KUKA KRL program: nutweldroutines.src, nutweldroutines.dat

--- nutweldroutines.src ---
&ACCESS RVO3
&REL 3482
&PARAM DISKPATH = KRC:\R1\TP\NutWeld
DEF NutWeldRoutines( )
   ;*********************************
   ;* Package:     NutWeldRoutines  *
   ;* Release      V1.0.4           *
   ;* Date:        01.2016          *
   ;* GUI Version: > = V8.3         *
   ;*********************************
   ; Declare in NutWeldData.dat Line 460:
   ;DECL REAL rSetUpperLVDT_CLS_W_NUT[3]
   ;rSetUpperLVDT_CLS_W_NUT[1] = 0.0
   ;rSetUpperLVDT_CLS_W_NUT[2] = 0.0
   ;rSetUpperLVDT_CLS_W_NUT[3] = 0.0
   ;DECL REAL rSetLowerLVDT_CLS_W_NUT[3]
   ;rSetLowerLVDT_CLS_W_NUT[1]  = 0.0
   ;rSetLowerLVDT_CLS_W_NUT[2]  = 0.0
   ;rSetLowerLVDT_CLS_W_NUT[3]  = 0.0
   ;DECL BOOL bSaveCurrentValue1=FALSE
   ;DECL BOOL bSaveCurrentValue2=FALSE
   ;DECL BOOL bSaveCurrentValue3=FALSE
END

GLOBAL DEF NutWeld_Bkg( )
   ;FOLD Details
      ;FOLD Declaration
         DECL REAL rPrimaryValue, rSecondaryValue, rSensorSample
         DECL INT nStepCnt
         DECL BOOL bSensorRetry
      ;ENDFOLD (Declaration)
      ;FOLD Implementation
         dopw1_Hidraulyc_Valve = ($PERI_RDY==TRUE)
         dopw2_Hidraulyc_Valve = (($PERI_RDY==TRUE) AND (nMaxGunNr>=2))
         dopw3_Hidraulyc_Valve = (($PERI_RDY==TRUE) AND (nMaxGunNr>=3))
         IF (($EXT==TRUE) AND (bNutWeld_InhibitWeld==TRUE)) THEN
            bNutWeld_InhibitWeld=FALSE ; Weld Inhibit not allowed in Auto
            nNutWeld_Handle_SPS=Set_Krlmsg (#NOTIFY, NutWeld_Msg[60], NutWeld_MsgPar[], NutWeld_MsgOpt_NoStop)
         ENDIF
         ;FOLD Program Reset/Cancel
            IF ((($PRO_STATE1==#P_FREE) OR ($PRO_STATE1==#P_RESET)) AND (bNutWeldProcessReset==FALSE)) THEN
               bNutWeldProcessReset=TRUE
               NutWeld_ProcessReset( )
            ELSE
               IF (($PRO_STATE1<>#P_FREE) AND ($PRO_STATE1<>#P_RESET)) THEN
                  bNutWeldProcessReset=FALSE
               ENDIF
            ENDIF
         ;ENDFOLD (Program Reset/Cancel)
         ;FOLD Status Key Control
            ;FOLD USKB1 - Process Control
               bNutWeldWOJoining = ((($MODE_OP==#EX) AND (di004UseDryCycle==TRUE)) OR ((($MODE_OP==#T1) OR ($MODE_OP==#T2)) AND (bNutWeldWOJoinSTK==TRUE)))
               IF (($MODE_OP==#T1) OR ($MODE_OP==#T2)) THEN
                  IF ((bNutWeldResetSTK==TRUE) AND ($OUT[Get_FaultResetNr(nNutWeldGunNrSTK)]==FALSE)) THEN
                     bNutWeldResetSTK=FALSE
                     PULSE($OUT[Get_FaultResetNr(nNutWeldGunNrSTK)],TRUE,0.25)
                  ENDIF
               ENDIF
            ;ENDFOLD (USKB1 - Process Control)
            ;FOLD USKB2 - Manual Control
               IF (bNutWeldOpnGunSTK==TRUE) THEN
                  dopw_GunWork(nNutWeldGunNrSTK,FALSE)
                  bNutWeldOpnGunSTK=FALSE
               ENDIF
               IF (bNutWeldClsGunSTK==TRUE) THEN
                  dopw_GunWork(nNutWeldGunNrSTK,TRUE)
                  bNutWeldClsGunSTK=FALSE
               ENDIF
               IF (bNutWeldAdvRetPinSTK==TRUE) THEN
                  dopw_PinAdv(nNutWeldGunNrSTK,dipw_PinReturn(nNutWeldGunNrSTK))
                  bNutWeldAdvRetPinSTK=FALSE
               ENDIF
            ;ENDFOLD (USKB2 - Manual Control)
            ;FOLD USKB3-4 Manual NutWeld
               IF ((bNutWeld_ManWeld_Active==TRUE) AND (bNutWeld_ManWeld_Step[20]==TRUE)) THEN
                  bNutWeld_ManWeld_Active=FALSE
                  bNutWeldManWeldSTK=FALSE
                  dopw_GunWork(nNutWeldGunNrSTK,FALSE)
                  dopw_WeldInit(nNutWeldGunNrSTK,FALSE)
                  dopw_NutIntensify(nNutWeldGunNrSTK,FALSE)
                  dopw_StartFeed(nNutWeldGunNrSTK,FALSE)
                  dopw_SetPrgNr(nNutWeldGunNrSTK, 0 )
                  $TIMER_STOP[nNutWeldManWeldTmr]=TRUE
                  FOR nStepCnt=1 to 20
                     bNutWeld_ManWeld_Step[nStepCnt]=FALSE
                  ENDFOR
               ENDIF
               IF ((bNutWeld_ManWeld_Active==TRUE) AND (bNutWeld_ManWeld_Step[11]==TRUE) AND (bNutWeld_ManWeld_Step[12]==FALSE)) THEN
                  ; Open Gun
                  dopw_GunWork(nNutWeldGunNrSTK,FALSE)
                  bNutWeld_ManWeld_Step[20]=TRUE ; Reset Process
               ENDIF
               IF ((bNutWeld_ManWeld_Active==TRUE) AND (bNutWeld_ManWeld_Step[10]==TRUE) AND (bNutWeld_ManWeld_Step[11]==FALSE)) THEN
                  ; Check for Weld Complete
                  IF ($TIMER_FLAG[nNutWeldManWeldTmr]==TRUE) THEN
                     bNutWeld_ManWeld_Step[20]=TRUE ; Reset Process
                     nNutWeld_Handle_SPS=Set_Krlmsg (#NOTIFY, NutWeld_Msg[19], NutWeld_MsgPar[], NutWeld_MsgOpt_NoStop)
                  ELSE
                     IF (dipw_WeldComplete(nNutWeldGunNrSTK)==TRUE) THEN
                        dopw_WeldInit(nNutWeldGunNrSTK,FALSE)
                        dopw_NutIntensify(nNutWeldGunNrSTK,FALSE)
                        bNutWeld_ManWeld_Step[11]=TRUE
                     ENDIF
                  ENDIF
               ENDIF
               IF ((bNutWeld_ManWeld_Active==TRUE) AND (bNutWeld_ManWeld_Step[9]==TRUE) AND (bNutWeld_ManWeld_Step[10]==FALSE)) THEN
                  ; Weld Initiate
                  dopw_WeldInit(nNutWeldGunNrSTK,TRUE)
                  bNutWeld_ManWeld_Step[10]=TRUE
               ENDIF
               IF ((bNutWeld_ManWeld_Active==TRUE) AND (bNutWeld_ManWeld_Step[8]==TRUE) AND (bNutWeld_ManWeld_Step[9]==FALSE)) THEN
                  ; Intensify Gun
                  dopw_NutIntensify(nNutWeldGunNrSTK,TRUE)
                  ; Check for Gun intensified
                  IF ($TIMER_FLAG[nNutWeldManWeldTmr]==TRUE) THEN
                     bNutWeld_ManWeld_Step[20]=TRUE ; Reset Process
                     nNutWeld_Handle_SPS=Set_Krlmsg (#NOTIFY, NutWeld_Msg[18], NutWeld_MsgPar[], NutWeld_MsgOpt_NoStop)
                  ELSE
                     IF (dipw_IntensfPresOk(nNutWeldGunNrSTK)==TRUE) THEN
                        bNutWeld_ManWeld_Step[9]=TRUE
                     ENDIF
                  ENDIF
               ENDIF
               IF ((bNutWeld_ManWeld_Active==TRUE) AND (bNutWeld_ManWeld_Step[7]==TRUE) AND (bNutWeld_ManWeld_Step[8]==FALSE)) THEN
                  ; Check for Nut Present
                  bSensorRetry=FALSE
                  IF (bByPassSmartelec==TRUE) THEN
                     bNutWeld_ManWeld_Step[8]=TRUE
                  ELSE
                     IF ($TIMER_FLAG[nNutWeldManWeldTmr]==TRUE) THEN
                        bNutWeld_ManWeld_Step[20]=TRUE ; Reset Process
                        nNutWeld_Handle_SPS=Set_Krlmsg (#NOTIFY, NutWeld_Msg[nManWeldFault], NutWeld_MsgPar[], NutWeld_MsgOpt_NoStop)
                     ELSE
                        rPrimaryValue = ABS(aiNutSensor(nNutWeldGunNrSTK));
                        WAIT SEC rSensorSettleTime;
                        rSecondaryValue = ABS(aiNutSensor(nNutWeldGunNrSTK));
                        IF (ABS(rPrimaryValue - rSecondaryValue) <= 2) THEN
                           rSensorSample=ABS(aiNutSensor(nNutWeldGunNrSTK))
                           IF ((rSensorSample <= (rNutInvertedValueInUse + rNutSensorTolInUse)) AND (rSensorSample >= (rNutInvertedValueInUse - rNutSensorTolInUse))) THEN
                              nManWeldFault=55
                              bSensorRetry=TRUE
                           ENDIF
                           IF ((rSensorSample <= (rNoNutValueInUse + rNutSensorTolInUse)) AND (rSensorSample >= (rNoNutValueInUse - rNutSensorTolInUse)) AND (bSensorRetry == FALSE)) THEN
                              nManWeldFault=54
                              bSensorRetry=TRUE
                           ENDIF
                           IF ((rSensorSample <= (rNutPresentValueInUse - rNutSensorTol2InUse)) AND (bSensorRetry == FALSE)) THEN
                              nManWeldFault=56
                              bSensorRetry=TRUE
                           ENDIF
                           IF (bSensorRetry==FALSE) THEN
                              nManWeldFault=0
                              bNutWeld_ManWeld_Step[8]=TRUE
                           ENDIF
                        ENDIF
                     ENDIF
                  ENDIF
               ENDIF
               IF ((bNutWeld_ManWeld_Active==TRUE) AND (bNutWeld_ManWeld_Step[6]==TRUE) AND (bNutWeld_ManWeld_Step[7]==FALSE)) THEN
                  ; Check for Gun Closed
                  IF ($TIMER_FLAG[nNutWeldManWeldTmr]==TRUE) THEN
                     bNutWeld_ManWeld_Step[20]=TRUE ; Reset Process
                     nNutWeld_Handle_SPS=Set_Krlmsg (#NOTIFY, NutWeld_Msg[35], NutWeld_MsgPar[], NutWeld_MsgOpt_NoStop)
                  ELSE
                     IF (bpw_GunAtWork(nNutWeldGunNrSTK)==TRUE) THEN
                        bNutWeld_ManWeld_Step[7]=TRUE
                     ENDIF
                  ENDIF
               ENDIF
               IF ((bNutWeld_ManWeld_Active==TRUE) AND (bNutWeld_ManWeld_Step[5]==TRUE) AND (bNutWeld_ManWeld_Step[6]==FALSE)) THEN
                  ; Check for Nut Fed
                  IF ($TIMER_FLAG[nNutWeldManWeldTmr]==TRUE) THEN
                     bNutWeld_ManWeld_Step[20]=TRUE ; Reset Process
                     nNutWeld_Handle_SPS=Set_Krlmsg (#NOTIFY, NutWeld_Msg[49], NutWeld_MsgPar[], NutWeld_MsgOpt_NoStop)
                     dopw_StartFeed(nNutWeldGunNrSTK,FALSE)
                  ELSE
                     IF (dipw_FeedComplt(nNutWeldGunNrSTK)==TRUE) THEN
                        bNutWeld_ManWeld_Step[6]=TRUE
                        ; Close the gun
                        dopw_StartFeed(nNutWeldGunNrSTK,FALSE)
                        dopw_NutIntensify(nNutWeldGunNrSTK,FALSE)
                        dopw_GunWork(nNutWeldGunNrSTK,TRUE)
                     ENDIF
                  ENDIF
               ENDIF
               IF ((bNutWeld_ManWeld_Active==TRUE) AND (bNutWeld_ManWeld_Step[4]==TRUE) AND (bNutWeld_ManWeld_Step[5]==FALSE)) THEN
                  ; Feed a Nut
                  dopw_StartFeed(nNutWeldGunNrSTK,TRUE)
                  bNutWeld_ManWeld_Step[5]=TRUE
               ENDIF
               IF ((bNutWeld_ManWeld_Active==TRUE) AND (bNutWeld_ManWeld_Step[3]==TRUE) AND (bNutWeld_ManWeld_Step[4]==FALSE)) THEN
                  ; Check for start conditions
                  IF (dipw_XtfmrTempOk(nNutWeldGunNrSTK)==FALSE) THEN
                     bNutWeld_ManWeld_Step[20]=TRUE ; Reset Process
                     nNutWeld_Handle_SPS=Set_Krlmsg (#NOTIFY, NutWeld_Msg[50], NutWeld_MsgPar[], NutWeld_MsgOpt_NoStop)
                  ENDIF
                  IF (dipw_WaterOk(nNutWeldGunNrSTK)==FALSE) THEN
                     bNutWeld_ManWeld_Step[20]=TRUE ; Reset Process
                     nNutWeld_Handle_SPS=Set_Krlmsg (#NOTIFY, NutWeld_Msg[5], NutWeld_MsgPar[], NutWeld_MsgOpt_NoStop)
                  ENDIF
                  IF (dipw_IntensfPresOk(nNutWeldGunNrSTK)==TRUE) THEN
                     bNutWeld_ManWeld_Step[20]=TRUE ; Reset Process
                     nNutWeld_Handle_SPS=Set_Krlmsg (#NOTIFY, NutWeld_Msg[7], NutWeld_MsgPar[], NutWeld_MsgOpt_NoStop)
                  ENDIF
                  IF (dipw_Ready(nNutWeldGunNrSTK)==FALSE) THEN
                     bNutWeld_ManWeld_Step[20]=TRUE ; Reset Process
                     nNutWeld_Handle_SPS=Set_Krlmsg (#NOTIFY, NutWeld_Msg[8], NutWeld_MsgPar[], NutWeld_MsgOpt_NoStop)
                  ENDIF
                  IF (dipw_Fault(nNutWeldGunNrSTK)==TRUE) THEN
                     bNutWeld_ManWeld_Step[20]=TRUE ; Reset Process
                     nNutWeld_Handle_SPS=Set_Krlmsg (#NOTIFY, NutWeld_Msg[9], NutWeld_MsgPar[], NutWeld_MsgOpt_NoStop)
                  ENDIF
                  IF (dipw_SpearHome(nNutWeldGunNrSTK)==FALSE) THEN
                     bNutWeld_ManWeld_Step[20]=TRUE ; Reset Process
                     nNutWeld_Handle_SPS=Set_Krlmsg (#NOTIFY, NutWeld_Msg[47], NutWeld_MsgPar[], NutWeld_MsgOpt_NoStop)
                  ENDIF
                  IF (dipw_PinReturn(nNutWeldGunNrSTK)==FALSE) THEN
                     bNutWeld_ManWeld_Step[20]=TRUE ; Reset Process
                     nNutWeld_Handle_SPS=Set_Krlmsg (#NOTIFY, NutWeld_Msg[15], NutWeld_MsgPar[], NutWeld_MsgOpt_NoStop)
                  ENDIF
                  IF (bpw_GunAtHome(nNutWeldGunNrSTK)==FALSE) THEN
                     bNutWeld_ManWeld_Step[20]=TRUE ; Reset Process
                     nNutWeld_Handle_SPS=Set_Krlmsg (#NOTIFY, NutWeld_Msg[51], NutWeld_MsgPar[], NutWeld_MsgOpt_NoStop)
                  ENDIF
                  bNutWeld_ManWeld_Step[4]=TRUE
               ENDIF
               IF ((bNutWeld_ManWeld_Active==TRUE) AND (bNutWeld_ManWeld_Step[2]==TRUE) AND (bNutWeld_ManWeld_Step[3]==FALSE)) THEN
                  IF (Exists_KrlDlg(nNutWeld_MWHandle, nNutWeld_MWKey)==FALSE) THEN
                     IF (nNutWeld_MWKey==1) THEN
                        bNutWeld_ManWeld_Step[3]=TRUE
                        dopw_SetPrgNr(nNutWeldGunNrSTK, nNutWeldSpotNrSTK )
                     ELSE
                        bNutWeld_ManWeld_Step[20]=TRUE ; Reset Process
                     ENDIF
                  ENDIF
                  nNutWeld_MWKey=0
               ENDIF
               IF ((bNutWeld_ManWeld_Active==TRUE) AND (bNutWeld_ManWeld_Step[1]==TRUE) AND (bNutWeld_ManWeld_Step[2]==FALSE)) THEN
                  bNutWeld_ManWeld_Step[2]=TRUE
                  NutWeld_MsgPar[1]={par_type #value, par_int 0}
                  NutWeld_MsgPar[1].par_int=nNutWeldGunNrSTK
                  NutWeld_MsgPar[2]={par_type #value, par_int 0}
                  NutWeld_MsgPar[2].par_int=nNutWeldSpotNrSTK
                  nNutWeld_MWHandle = Set_KrlDlg (NutWeld_Msg[34], NutWeld_MsgPar[], NutWeld_SK_OKCancel[], NutWeld_MsgOpt_NoStop)
               ENDIF
               IF ((bNutWeldManWeldSTK==TRUE) AND (bNutWeld_ManWeld_Step[1]==FALSE)) THEN
                  IF (bNutWeldWOJoining==FALSE) THEN
                     bNutWeld_ManWeld_Active=TRUE
                     bNutWeld_ManWeld_Step[1]=TRUE
                     dopw_GunWork(nNutWeldGunNrSTK,FALSE)
                     dopw_StartFeed(nNutWeldGunNrSTK,FALSE)
                     dopw_WeldInit(nNutWeldGunNrSTK,FALSE)
                     dopw_NutIntensify(nNutWeldGunNrSTK,FALSE)
                     NutWeldManual.GunNr=nNutWeldGunNrSTK
                     NutWeldManual.SpotNr=nNutWeldSpotNrSTK
                     PWInitUserIO(NutWeldManual)
                     $TIMER_STOP[nNutWeldManWeldTmr]=TRUE
                     $TIMER[nNutWeldManWeldTmr]=(nNutWeld_ManWeld_Timeout*(-1000))
                     $TIMER_STOP[nNutWeldManWeldTmr]=FALSE
                  ELSE
                     nNutWeld_Handle_SPS=Set_Krlmsg (#NOTIFY, NutWeld_Msg[33], NutWeld_MsgPar[], NutWeld_MsgOpt_NoStop)
                     bNutWeldManWeldSTK=FALSE
                  ENDIF
               ENDIF
            ;ENDFOLD (USKB3-4 Manual NutWeld)
            ;FOLD USKB4 - Gun Maintenance Actions
               ;FOLD USKB4-2 Test Gun Force
                  IF ((bNutWeld_TstFrce_Active==TRUE) AND (bNutWeld_TstFrce_Step[10]==TRUE)) THEN
                     bNutWeld_TstFrce_Active=FALSE
                     bNutWeldTstFrceSTK=FALSE
                     dopw_GunWork(nNutWeldGunNrSTK,FALSE)
                     dopw_WeldInit(nNutWeldGunNrSTK,FALSE)
                     dopw_NutIntensify(nNutWeldGunNrSTK,FALSE)
                     dopw_SetPrgNr(nNutWeldGunNrSTK, 0)
                     $TIMER_STOP[nNutWeldManWeldTmr]=TRUE
                     $TIMER_STOP[nNutWeldSignalTmr]=TRUE
                     $TIMER[nNutWeldManWeldTmr]=-1000
                     $TIMER[nNutWeldSignalTmr]=-750
                     FOR nStepCnt=1 to 10
                        bNutWeld_TstFrce_Step[nStepCnt]=FALSE
                     ENDFOR
                  ENDIF
                  IF ((bNutWeld_TstFrce_Active==TRUE) AND (bNutWeld_TstFrce_Step[6]==TRUE) AND (bNutWeld_TstFrce_Step[7]==FALSE)) THEN
                     ; Wait Intensify Time
                     IF ($TIMER_FLAG[nNutWeldSignalTmr]==TRUE) THEN
                        $TIMER_STOP[nNutWeldSignalTmr]=TRUE
                        $TIMER[nNutWeldSignalTmr]=(-2000)
                        dopw_NutIntensify(nNutWeldGunNrSTK,FALSE)
                        dopw_GunWork(nNutWeldGunNrSTK,FALSE)
                        bNutWeld_TstFrce_Step[10]=TRUE
                        NutWeld_MsgPar[1]={par_type #value, par_int 0}
                        NutWeld_MsgPar[1].par_int=nNutWeldGunNrSTK
                        nNutWeld_Handle_SPS=Set_Krlmsg (#NOTIFY, NutWeld_Msg[44], NutWeld_MsgPar[], NutWeld_MsgOpt_NoStop)
                     ENDIF
                  ENDIF
                  IF ((bNutWeld_TstFrce_Active==TRUE) AND (bNutWeld_TstFrce_Step[5]==TRUE) AND (bNutWeld_TstFrce_Step[6]==FALSE)) THEN
                     ; Check for Gun Closed
                     IF (($TIMER_FLAG[nNutWeldManWeldTmr]==TRUE) AND (bpw_GunAtHome(nNutWeldGunNrSTK)==TRUE)) THEN
                        bNutWeld_TstFrce_Step[10]=TRUE ; Reset Process
                        nNutWeld_Handle_SPS=Set_Krlmsg (#NOTIFY, NutWeld_Msg[35], NutWeld_MsgPar[], NutWeld_MsgOpt_NoStop)
                     ELSE
                        IF (($TIMER_FLAG[nNutWeldSignalTmr]==TRUE) AND (bpw_GunAtHome(nNutWeldGunNrSTK)==FALSE)) THEN
                           ; Intensify Gun
                           dopw_NutIntensify(nNutWeldGunNrSTK,TRUE)
                           $TIMER_STOP[nNutWeldSignalTmr]=TRUE
                           $TIMER[nNutWeldSignalTmr]=(-2000)
                           $TIMER_STOP[nNutWeldSignalTmr]=FALSE
                           bNutWeld_TstFrce_Step[6]=TRUE
                        ENDIF
                     ENDIF
                  ENDIF
                  IF ((bNutWeld_TstFrce_Active==TRUE) AND (bNutWeld_TstFrce_Step[4]==TRUE) AND (bNutWeld_TstFrce_Step[5]==FALSE)) THEN
                     IF (Exists_KrlDlg(nNutWeld_TFHandle, nNutWeld_TFKey)==FALSE) THEN
                        IF (nNutWeld_TFKey==1) THEN
                           $TIMER_STOP[nNutWeldManWeldTmr]=FALSE
                           dopw_NutIntensify(nNutWeldGunNrSTK,FALSE)
                           dopw_GunWork(nNutWeldGunNrSTK,TRUE)
                           $TIMER_STOP[nNutWeldSignalTmr]=TRUE
                           $TIMER[nNutWeldSignalTmr]=(-2000)
                           $TIMER_STOP[nNutWeldSignalTmr]=FALSE
                           bNutWeld_TstFrce_Step[5]=TRUE
                        ELSE
                           bNutWeld_TstFrce_Step[10]=TRUE ; Reset Process
                        ENDIF
                     ENDIF
                     nNutWeld_TFKey=0
                  ENDIF
                  IF ((bNutWeldTstFrceSTK==TRUE) AND (bNutWeld_TstFrce_Step[3]==TRUE) AND (bNutWeld_TstFrce_Step[4]==FALSE)) THEN
                     bNutWeld_TstFrce_Active=TRUE
                     bNutWeld_TstFrce_Step[4]=TRUE
                     $TIMER_STOP[nNutWeldManWeldTmr]=TRUE
                     $TIMER[nNutWeldManWeldTmr]=(nNutWeld_ManWeld_Timeout*(-1000))
                     nNutWeld_TFKey=0
                     NutWeld_MsgPar[1]={par_type #value, par_int 0}
                     NutWeld_MsgPar[1].par_int=nNutWeldGunNrSTK
                     nNutWeld_TFHandle = Set_KrlDlg (NutWeld_Msg[38], NutWeld_MsgPar[], NutWeld_SK_TstCncl[], NutWeld_MsgOpt_NoStop)
                  ENDIF
                  IF ((bNutWeld_TstFrce_Active==TRUE) AND (bNutWeld_TstFrce_Step[2]==TRUE) AND (bNutWeld_TstFrce_Step[3]==FALSE)) THEN
                     ; Check for Gun Home
                     IF ($TIMER_FLAG[nNutWeldManWeldTmr]==TRUE) THEN
                        bNutWeld_TstFrce_Step[10]=TRUE ; Reset Process
                        nNutWeld_Handle_SPS=Set_Krlmsg (#NOTIFY, NutWeld_Msg[32], NutWeld_MsgPar[], NutWeld_MsgOpt_NoStop)
                     ELSE
                        IF (($TIMER_FLAG[nNutWeldSignalTmr]==FALSE) AND (bpw_GunAtHome(nNutWeldGunNrSTK)==TRUE)) THEN
                           ; Intensify Gun
                           $TIMER_STOP[nNutWeldSignalTmr]=TRUE
                           $TIMER[nNutWeldSignalTmr]=(-2000)
                           bNutWeld_TstFrce_Step[3]=TRUE
                        ENDIF
                     ENDIF
                  ENDIF
                  IF ((bNutWeld_TstFrce_Active==TRUE) AND (bNutWeld_TstFrce_Step[1]==TRUE) AND (bNutWeld_TstFrce_Step[2]==FALSE)) THEN
                     IF (Exists_KrlDlg(nNutWeld_TFHandle, nNutWeld_TFKey)==FALSE) THEN
                        IF (nNutWeld_TFKey==1) THEN
                           dopw_NutIntensify(nNutWeldGunNrSTK,FALSE)
                           dopw_GunWork(nNutWeldGunNrSTK,FALSE)
                           $TIMER_STOP[nNutWeldSignalTmr]=TRUE
                           $TIMER[nNutWeldSignalTmr]=(-3000)
                           $TIMER_STOP[nNutWeldSignalTmr]=FALSE
                           bNutWeld_TstFrce_Step[2]=TRUE
                        ELSE
                           bNutWeld_TstFrce_Step[10]=TRUE ; Reset Process
                        ENDIF
                     ENDIF
                     nNutWeld_TFKey=0
                  ENDIF
                  IF ((bNutWeldTstFrceSTK==TRUE) AND (bNutWeld_TstFrce_Step[1]==FALSE) AND (bpw_GunAtHome(nNutWeldGunNrSTK )==TRUE)) THEN
                     bNutWeld_TstFrce_Active=TRUE
                     bNutWeld_TstFrce_Step[1]=TRUE
                     bNutWeld_TstFrce_Step[2]=TRUE
                     bNutWeld_TstFrce_Step[3]=TRUE
                     nNutWeld_TFKey=0
                  ELSE
                     IF ((bNutWeldTstFrceSTK==TRUE) AND (bNutWeld_TstFrce_Step[1]==FALSE) AND (bpw_GunAtHome(nNutWeldGunNrSTK )==FALSE)) THEN
                        bNutWeld_TstFrce_Active=TRUE
                        bNutWeld_TstFrce_Step[1]=TRUE
                        nNutWeld_TFKey=0
                        NutWeld_MsgPar[1]={par_type #value, par_int 0}
                        NutWeld_MsgPar[1].par_int=nNutWeldGunNrSTK
                        nNutWeld_TFHandle = Set_KrlDlg (NutWeld_Msg[51], NutWeld_MsgPar[], NutWeld_SK_HomeGun[], NutWeld_MsgOpt_NoStop)
                        $TIMER_STOP[nNutWeldManWeldTmr]=TRUE
                        $TIMER[nNutWeldManWeldTmr]=(nNutWeld_ManWeld_Timeout*(-1000))
                     ENDIF
                  ENDIF
               ;ENDFOLD (USKB4-2 Test Gun Force)
               ;FOLD USKB4-3 Teach Analog
                  ;FOLD USKB4-2.4 Check
                     IF ((bNutWeld_AlgCheck_Active==TRUE) AND (bNutWeld_AlgCheck_Step[10]==TRUE)) THEN
                        bNutWeld_AlgCheck_Active=FALSE
                        bNutWeldAlgCheckReq=FALSE
                        FOR nStepCnt=1 to 10
                           bNutWeld_AlgCheck_Step[nStepCnt]=FALSE
                        ENDFOR
                        bNutWeld_TchAnlg_Active=FALSE
                        bNutWeldTchAnlgSTK=TRUE
                        FOR nStepCnt=1 to 10
                           bNutWeld_TchAnlg_Step[nStepCnt]=FALSE
                        ENDFOR
                     ENDIF
                     IF ((bNutWeld_AlgCheck_Active==TRUE) AND (bNutWeld_AlgCheck_Step[8]==TRUE) AND (bNutWeld_AlgCheck_Step[9]==FALSE)) THEN
                        IF (Exists_KrlDlg(nNutWeld_TA4Handle, nNutWeld_TA4Key)==FALSE) THEN
                           IF (nNutWeld_TA4Key==1) THEN
                              nNutWeld_TA4Key=0
                              bNutWeld_AlgCheck_Step[9]=TRUE
                              bNutWeld_AlgCheck_Step[10]=TRUE
                           ELSE
                              bNutWeld_AlgCheck_Step[10]=TRUE ; Reset Process
                           ENDIF
                        ENDIF
                        nNutWeld_TA4Key=0
                     ENDIF
                     IF ((bNutWeld_AlgCheck_Active==TRUE) AND (bNutWeld_AlgCheck_Step[7]==TRUE) AND (bNutWeld_AlgCheck_Step[8]==FALSE)) THEN
                        IF (rNutInvertedValue[nNutWeldGunNrSTK] < (rNutPresentValue[nNutWeldGunNrSTK] + rNutSensorTolerance[nNutWeldGunNrSTK])) THEN
                           nNutWeld_TA4Handle = Set_KrlDlg (NutWeld_Msg[59], NutWeld_MsgPar[], NutWeld_SK_Next[], NutWeld_MsgOpt_NoStop)
                           bNutWeld_AlgCheck_Step[8]=TRUE
                        ELSE
                           bNutWeld_AlgCheck_Step[10]=TRUE
                        ENDIF
                     ENDIF
                     IF ((bNutWeld_AlgCheck_Active==TRUE) AND (bNutWeld_AlgCheck_Step[6]==TRUE) AND (bNutWeld_AlgCheck_Step[7]==FALSE)) THEN
                        IF (Exists_KrlDlg(nNutWeld_TA4Handle, nNutWeld_TA4Key)==FALSE) THEN
                           IF (nNutWeld_TA4Key==1) THEN
                              nNutWeld_TA4Key=0
                              bNutWeld_AlgCheck_Step[7]=TRUE
                           ELSE
                              bNutWeld_AlgCheck_Step[10]=TRUE ; Reset Process
                           ENDIF
                        ENDIF
                        nNutWeld_TA4Key=0
                     ENDIF
                     IF ((bNutWeld_AlgCheck_Active==TRUE) AND (bNutWeld_AlgCheck_Step[5]==TRUE) AND (bNutWeld_AlgCheck_Step[6]==FALSE)) THEN
                        IF (Exists_KrlDlg(nNutWeld_TA4Handle, nNutWeld_TA4Key)==FALSE) THEN
                           IF (nNutWeld_TA4Key==1) THEN
                              nNutWeld_TA4Key=0
                              bNutWeld_AlgCheck_Step[6]=TRUE
                              IF (rNoNutValue[nNutWeldGunNrSTK] > (rNutPresentValue[nNutWeldGunNrSTK] - rNutSensorTolerance[nNutWeldGunNrSTK])) THEN
                                 nNutWeld_TA4Handle = Set_KrlDlg (NutWeld_Msg[58], NutWeld_MsgPar[], NutWeld_SK_Next[], NutWeld_MsgOpt_NoStop)
                              ELSE
                                 bNutWeld_AlgCheck_Step[7]=TRUE
                              ENDIF
                           ELSE
                              bNutWeld_AlgCheck_Step[10]=TRUE ; Reset Process
                           ENDIF
                        ENDIF
                        nNutWeld_TA4Key=0
                     ENDIF
                     IF ((bNutWeld_AlgCheck_Active==TRUE) AND (bNutWeld_AlgCheck_Step[4]==TRUE) AND (bNutWeld_AlgCheck_Step[5]==FALSE)) THEN
                        IF (Exists_KrlDlg(nNutWeld_TA4Handle, nNutWeld_TA4Key)==FALSE) THEN
                           IF (nNutWeld_TA4Key==1) THEN
                              nNutWeld_TA4Key=0
                              NutWeld_MsgPar[1].par_real=rNutInvertedValue[nNutWeldGunNrSTK]
                              nNutWeld_TA4Handle = Set_KrlDlg (NutWeld_Msg[57], NutWeld_MsgPar[], NutWeld_SK_Next[], NutWeld_MsgOpt_NoStop)
                              bNutWeld_AlgCheck_Step[5]=TRUE
                           ELSE
                              bNutWeld_AlgCheck_Step[10]=TRUE ; Reset Process
                           ENDIF
                        ENDIF
                        nNutWeld_TA4Key=0
                     ENDIF
                     IF ((bNutWeld_AlgCheck_Active==TRUE) AND (bNutWeld_AlgCheck_Step[3]==TRUE) AND (bNutWeld_AlgCheck_Step[4]==FALSE)) THEN
                        IF (Exists_KrlDlg(nNutWeld_TA4Handle, nNutWeld_TA4Key)==FALSE) THEN
                           IF (nNutWeld_TA4Key==1) THEN
                              nNutWeld_TA4Key=0
                              NutWeld_MsgPar[1].par_real=rNutPresentValue[nNutWeldGunNrSTK]
                              nNutWeld_TA4Handle = Set_KrlDlg (NutWeld_Msg[31], NutWeld_MsgPar[], NutWeld_SK_Next[], NutWeld_MsgOpt_NoStop)
                              bNutWeld_AlgCheck_Step[4]=TRUE
                           ELSE
                              bNutWeld_AlgCheck_Step[10]=TRUE ; Reset Process
                           ENDIF
                        ENDIF
                        nNutWeld_TA4Key=0
                     ENDIF
                     IF ((bNutWeld_AlgCheck_Active==TRUE) AND (bNutWeld_AlgCheck_Step[2]==TRUE) AND (bNutWeld_AlgCheck_Step[3]==FALSE)) THEN
                        IF (Exists_KrlDlg(nNutWeld_TA4Handle, nNutWeld_TA4Key)==FALSE) THEN
                           IF (nNutWeld_TA4Key==1) THEN
                              nNutWeld_TA4Key=0
                              NutWeld_MsgPar[1].par_real=rNoNutValue[nNutWeldGunNrSTK]
                              nNutWeld_TA4Handle = Set_KrlDlg (NutWeld_Msg[30], NutWeld_MsgPar[], NutWeld_SK_Next[], NutWeld_MsgOpt_NoStop)
                              bNutWeld_AlgCheck_Step[3]=TRUE
                           ELSE
                              bNutWeld_AlgCheck_Step[10]=TRUE ; Reset Process
                           ENDIF
                        ENDIF
                        nNutWeld_TA4Key=0
                     ENDIF
                     IF ((bNutWeld_AlgCheck_Active==TRUE) AND (bNutWeld_AlgCheck_Step[1]==TRUE) AND (bNutWeld_AlgCheck_Step[2]==FALSE)) THEN
                        IF (Exists_KrlDlg(nNutWeld_TA4Handle, nNutWeld_TA4Key)==FALSE) THEN
                           IF (nNutWeld_TA4Key==1) THEN
                              nNutWeld_TA4Key=0
                              NutWeld_MsgPar[1]={par_type #value, par_real 0}
                              NutWeld_MsgPar[1].par_real=rNutSensorTolerance2[nNutWeldGunNrSTK]
                              nNutWeld_TA4Handle = Set_KrlDlg (NutWeld_Msg[29], NutWeld_MsgPar[], NutWeld_SK_Next[], NutWeld_MsgOpt_NoStop)
                              bNutWeld_AlgCheck_Step[2]=TRUE
                           ELSE
                              bNutWeld_AlgCheck_Step[10]=TRUE ; Reset Process
                           ENDIF
                        ENDIF
                        nNutWeld_TA4Key=0
                     ENDIF
                     IF ((bNutWeldAlgCheckReq==TRUE) AND (bNutWeld_AlgCheck_Step[1]==FALSE)) THEN
                        bNutWeld_AlgCheck_Active=TRUE
                        bNutWeld_AlgCheck_Step[1]=TRUE
                        nNutWeld_TA4Key=0
                        NutWeld_MsgPar[1]={par_type #value, par_real 0}
                        NutWeld_MsgPar[1].par_real=rNutSensorTolerance[nNutWeldGunNrSTK]
                        nNutWeld_TA4Handle = Set_KrlDlg (NutWeld_Msg[28], NutWeld_MsgPar[], NutWeld_SK_Next[], NutWeld_MsgOpt_NoStop)
                     ENDIF
                  ;ENDFOLD (USKB4-2.4 Check)
                  ;FOLD USKB4-2.3 Inverted Nut
                     IF ((bNutWeld_AlgInNut_Active==TRUE) AND (bNutWeld_AlgInNut_Step[10]==TRUE)) THEN
                        bNutWeld_AlgInNut_Active=FALSE
                        bNutWeldAlgInNutReq=FALSE
                        dopw_GunWork(nNutWeldGunNrSTK,FALSE)
                        dopw_NutIntensify(nNutWeldGunNrSTK,FALSE)
                        FOR nStepCnt=1 to 10
                           bNutWeld_AlgInNut_Step[nStepCnt]=FALSE
                        ENDFOR
                        bNutWeld_TchAnlg_Active=FALSE
                        bNutWeldTchAnlgSTK=TRUE
                        $TIMER_STOP[nNutWeldManWeldTmr]=TRUE
                        $TIMER_STOP[nNutWeldSignalTmr]=TRUE
                        $TIMER[nNutWeldManWeldTmr]=-1000
                        $TIMER[nNutWeldSignalTmr]=-750
                        FOR nStepCnt=1 to 10
                           bNutWeld_TchAnlg_Step[nStepCnt]=FALSE
                        ENDFOR
                     ENDIF
                     IF ((bNutWeld_AlgInNut_Active==TRUE) AND (bNutWeld_AlgInNut_Step[6]==TRUE) AND (bNutWeld_AlgInNut_Step[7]==FALSE)) THEN
                        bNutWeld_AlgInNut_Active=FALSE
                        bNutWeldAlgInNutReq=TRUE
                        FOR nStepCnt=1 to 10
                           bNutWeld_AlgInNut_Step[nStepCnt]=FALSE
                        ENDFOR
                     ENDIF
                     IF ((bNutWeld_AlgInNut_Active==TRUE) AND (bNutWeld_AlgInNut_Step[5]==TRUE) AND (bNutWeld_AlgInNut_Step[6]==FALSE)) THEN
                        IF (Exists_KrlDlg(nNutWeld_TA3Handle, nNutWeld_TA3Key)==FALSE) THEN
                           SWITCH nNutWeld_TA3Key
                              CASE 1 ; Accept - Store value and exit
                                 rNutInvertedValue[nNutWeldGunNrSTK]=rNutSensorValueTemp
                                 rNutSensorValueTemp=0.0
                                 bNutWeld_AlgInNut_Step[10]=TRUE ; Reset Process
                              CASE 2 ; Rerun - discard value and re-execute
                                 rNutSensorValueTemp=0.0
                                 bNutWeld_AlgInNut_Step[6]=TRUE ; Local Reset Process
                              CASE 3 ; Cancel - discard value and return to main selection
                                 rNutSensorValueTemp=0.0
                                 bNutWeld_AlgInNut_Step[10]=TRUE ; Reset Process
                           ENDSWITCH
                        ENDIF
                        nNutWeld_TA3Key=0
                     ENDIF
                     IF ((bNutWeld_AlgInNut_Active==TRUE) AND (bNutWeld_AlgInNut_Step[4]==TRUE) AND (bNutWeld_AlgInNut_Step[5]==FALSE)) THEN
                        rNutSensorValueTemp=ABS(aiNutSensor(nNutWeldGunNrSTK))
                        dopw_NutIntensify(nNutWeldGunNrSTK,FALSE)
                        dopw_GunWork(nNutWeldGunNrSTK,FALSE)
                        NutWeld_MsgPar[1]={par_type #value, par_real 0}
                        NutWeld_MsgPar[1].par_real=rNutSensorValueTemp
                        nNutWeld_TA3Handle = Set_KrlDlg (NutWeld_Msg[53], NutWeld_MsgPar[], NutWeld_SK_AcptRerun[], NutWeld_MsgOpt_NoStop)
                        bNutWeld_AlgInNut_Step[5]=TRUE
                     ENDIF
                     IF ((bNutWeld_AlgInNut_Active==TRUE) AND (bNutWeld_AlgInNut_Step[3]==TRUE) AND (bNutWeld_AlgInNut_Step[4]==FALSE)) THEN
                        ; Smart Electrode Dwell Time
                        IF ($TIMER_FLAG[nNutWeldManWeldTmr]==TRUE) THEN
                           $TIMER_STOP[nNutWeldSignalTmr]=TRUE
                           $TIMER[nNutWeldSignalTmr]=(-1000)
                           bNutWeld_AlgInNut_Step[4]=TRUE
                        ENDIF
                     ENDIF
                     IF ((bNutWeld_AlgInNut_Active==TRUE) AND (bNutWeld_AlgInNut_Step[2]==TRUE) AND (bNutWeld_AlgInNut_Step[3]==FALSE)) THEN
                        ; Check for Gun Closed
                        IF ($TIMER_FLAG[nNutWeldManWeldTmr]==TRUE) THEN
                           bNutWeld_AlgInNut_Step[10]=TRUE ; Reset Process
                           nNutWeld_Handle_SPS=Set_Krlmsg (#NOTIFY, NutWeld_Msg[35], NutWeld_MsgPar[], NutWeld_MsgOpt_NoStop)
                        ELSE
                           IF (bpw_GunAtHome(nNutWeldGunNrSTK)==FALSE) THEN
                              $TIMER_STOP[nNutWeldSignalTmr]=TRUE
                              $TIMER[nNutWeldSignalTmr]=(-1000)
                              $TIMER_STOP[nNutWeldSignalTmr]=FALSE
                              bNutWeld_AlgInNut_Step[3]=TRUE
                           ENDIF
                        ENDIF
                     ENDIF
                     IF ((bNutWeld_AlgInNut_Active==TRUE) AND (bNutWeld_AlgInNut_Step[1]==TRUE) AND (bNutWeld_AlgInNut_Step[2]==FALSE)) THEN
                        IF (Exists_KrlDlg(nNutWeld_TA3Handle, nNutWeld_TA3Key)==FALSE) THEN
                           IF (nNutWeld_TA3Key==1) THEN
                              $TIMER_STOP[nNutWeldManWeldTmr]=FALSE
                              dopw_NutIntensify(nNutWeldGunNrSTK,FALSE)
                              dopw_GunWork(nNutWeldGunNrSTK,TRUE)
                              $TIMER_STOP[nNutWeldSignalTmr]=TRUE
                              $TIMER[nNutWeldSignalTmr]=(-750)
                              $TIMER_STOP[nNutWeldSignalTmr]=FALSE
                              bNutWeld_AlgInNut_Step[2]=TRUE
                           ELSE
                              bNutWeld_AlgInNut_Step[10]=TRUE ; Reset Process
                           ENDIF
                        ENDIF
                        nNutWeld_TA3Key=0
                     ENDIF
                     IF ((bNutWeldAlgInNutReq==TRUE) AND (bNutWeld_AlgInNut_Step[1]==FALSE)) THEN
                        bNutWeld_AlgInNut_Active=TRUE
                        bNutWeld_AlgInNut_Step[1]=TRUE
                        dopw_NutIntensify(nNutWeldGunNrSTK,FALSE)
                        dopw_GunWork(nNutWeldGunNrSTK,FALSE)
                        $TIMER_STOP[nNutWeldManWeldTmr]=TRUE
                        $TIMER[nNutWeldManWeldTmr]=(nNutWeld_ManWeld_Timeout*(-1000))
                        $TIMER_STOP[nNutWeldManWeldTmr]=FALSE
                        nNutWeld_TA3Key=0
                        nNutWeld_TA3Handle = Set_KrlDlg (NutWeld_Msg[52], NutWeld_MsgPar[], NutWeld_SK_CloseNWGun[], NutWeld_MsgOpt_NoStop)
                     ENDIF
                  ;ENDFOLD (USKB4-2.3 Inverted Nut)
                  ;FOLD USKB4-2.2 With Nut
                     IF ((bNutWeld_AlgWNut_Active==TRUE) AND (bNutWeld_AlgWNut_Step[10]==TRUE)) THEN
                        bNutWeld_AlgWNut_Active=FALSE
                        bNutWeldAlgWNutReq=FALSE
                        dopw_GunWork(nNutWeldGunNrSTK,FALSE)
                        dopw_NutIntensify(nNutWeldGunNrSTK,FALSE)
                        FOR nStepCnt=1 to 10
                           bNutWeld_AlgWNut_Step[nStepCnt]=FALSE
                        ENDFOR
                        bNutWeld_TchAnlg_Active=FALSE
                        bNutWeldTchAnlgSTK=TRUE
                        $TIMER_STOP[nNutWeldManWeldTmr]=TRUE
                        $TIMER_STOP[nNutWeldSignalTmr]=TRUE
                        $TIMER[nNutWeldManWeldTmr]=-1000
                        $TIMER[nNutWeldSignalTmr]=-750
                        FOR nStepCnt=1 to 10
                           bNutWeld_TchAnlg_Step[nStepCnt]=FALSE
                        ENDFOR
                     ENDIF
                     IF ((bNutWeld_AlgWNut_Active==TRUE) AND (bNutWeld_AlgWNut_Step[6]==TRUE) AND (bNutWeld_AlgWNut_Step[7]==FALSE)) THEN
                        bNutWeld_AlgWNut_Active=FALSE
                        bNutWeldAlgWNutReq=TRUE
                        FOR nStepCnt=1 to 10
                           bNutWeld_AlgWNut_Step[nStepCnt]=FALSE
                        ENDFOR
                     ENDIF
                     IF ((bNutWeld_AlgWNut_Active==TRUE) AND (bNutWeld_AlgWNut_Step[5]==TRUE) AND (bNutWeld_AlgWNut_Step[6]==FALSE)) THEN
                        IF (Exists_KrlDlg(nNutWeld_TA2Handle, nNutWeld_TA2Key)==FALSE) THEN
                           SWITCH nNutWeld_TA2Key
                              CASE 1 ; Accept - Store value and exit
                                 rNutPresentValue[nNutWeldGunNrSTK]=rNutSensorValueTemp
                                 rNutSensorValueTemp=0.0
                                 bNutWeld_AlgWNut_Step[10]=TRUE ; Reset Process
                              CASE 2 ; Rerun - discard value and re-execute
                                 rNutSensorValueTemp=0.0
                                 bNutWeld_AlgWNut_Step[6]=TRUE ; Local Reset Process
                              CASE 3 ; Cancel - discard value and return to main selection
                                 rNutSensorValueTemp=0.0
                                 bNutWeld_AlgWNut_Step[10]=TRUE ; Reset Process
                           ENDSWITCH
                        ENDIF
                        nNutWeld_TA2Key=0
                     ENDIF
                     IF ((bNutWeld_AlgWNut_Active==TRUE) AND (bNutWeld_AlgWNut_Step[4]==TRUE) AND (bNutWeld_AlgWNut_Step[5]==FALSE)) THEN
                        rNutSensorValueTemp=ABS(aiNutSensor(nNutWeldGunNrSTK))
                        dopw_NutIntensify(nNutWeldGunNrSTK,FALSE)
                        dopw_GunWork(nNutWeldGunNrSTK,FALSE)
                        NutWeld_MsgPar[1]={par_type #value, par_real 0}
                        NutWeld_MsgPar[1].par_real=rNutSensorValueTemp
                        nNutWeld_TA2Handle = Set_KrlDlg (NutWeld_Msg[43], NutWeld_MsgPar[], NutWeld_SK_AcptRerun[], NutWeld_MsgOpt_NoStop)
                        bNutWeld_AlgWNut_Step[5]=TRUE
                     ENDIF
                     IF ((bNutWeld_AlgWNut_Active==TRUE) AND (bNutWeld_AlgWNut_Step[3]==TRUE) AND (bNutWeld_AlgWNut_Step[4]==FALSE)) THEN
                        ; Smart Electrode Dwell Time
                        IF ($TIMER_FLAG[nNutWeldManWeldTmr]==TRUE) THEN
                           $TIMER_STOP[nNutWeldSignalTmr]=TRUE
                           $TIMER[nNutWeldSignalTmr]=(-1000)
                           bNutWeld_AlgWNut_Step[4]=TRUE
                        ENDIF
                     ENDIF
                     IF ((bNutWeld_AlgWNut_Active==TRUE) AND (bNutWeld_AlgWNut_Step[2]==TRUE) AND (bNutWeld_AlgWNut_Step[3]==FALSE)) THEN
                        ; Check for Gun Closed
                        IF ($TIMER_FLAG[nNutWeldManWeldTmr]==TRUE) THEN
                           bNutWeld_AlgWNut_Step[10]=TRUE ; Reset Process
                           nNutWeld_Handle_SPS=Set_Krlmsg (#NOTIFY, NutWeld_Msg[35], NutWeld_MsgPar[], NutWeld_MsgOpt_NoStop)
                        ELSE
                           IF (bpw_GunAtHome(nNutWeldGunNrSTK)==FALSE) THEN
                              $TIMER_STOP[nNutWeldSignalTmr]=TRUE
                              $TIMER[nNutWeldSignalTmr]=(-1000)
                              $TIMER_STOP[nNutWeldSignalTmr]=FALSE
                              bNutWeld_AlgWNut_Step[3]=TRUE
                           ENDIF
                        ENDIF
                     ENDIF
                     IF ((bNutWeld_AlgWNut_Active==TRUE) AND (bNutWeld_AlgWNut_Step[1]==TRUE) AND (bNutWeld_AlgWNut_Step[2]==FALSE)) THEN
                        IF (Exists_KrlDlg(nNutWeld_TA2Handle, nNutWeld_TA2Key)==FALSE) THEN
                           IF (nNutWeld_TA2Key==1) THEN
                              $TIMER_STOP[nNutWeldManWeldTmr]=FALSE
                              dopw_NutIntensify(nNutWeldGunNrSTK,FALSE)
                              dopw_GunWork(nNutWeldGunNrSTK,TRUE)
                              $TIMER_STOP[nNutWeldSignalTmr]=TRUE
                              $TIMER[nNutWeldSignalTmr]=(-750)
                              $TIMER_STOP[nNutWeldSignalTmr]=FALSE
                              bNutWeld_AlgWNut_Step[2]=TRUE
                           ELSE
                              bNutWeld_AlgWNut_Step[10]=TRUE ; Reset Process
                           ENDIF
                        ENDIF
                        nNutWeld_TA2Key=0
                     ENDIF
                     IF ((bNutWeldAlgWNutReq==TRUE) AND (bNutWeld_AlgWNut_Step[1]==FALSE)) THEN
                        bNutWeld_AlgWNut_Active=TRUE
                        bNutWeld_AlgWNut_Step[1]=TRUE
                        dopw_NutIntensify(nNutWeldGunNrSTK,FALSE)
                        dopw_GunWork(nNutWeldGunNrSTK,FALSE)
                        $TIMER_STOP[nNutWeldManWeldTmr]=TRUE
                        $TIMER[nNutWeldManWeldTmr]=(nNutWeld_ManWeld_Timeout*(-1000))
                        $TIMER_STOP[nNutWeldManWeldTmr]=FALSE
                        nNutWeld_TA2Key=0
                        nNutWeld_TA2Handle = Set_KrlDlg (NutWeld_Msg[41], NutWeld_MsgPar[], NutWeld_SK_CloseNWGun[], NutWeld_MsgOpt_NoStop)
                     ENDIF
                  ;ENDFOLD (USKB4-2.2 With Nut)
                  ;FOLD USKB4-2.1 No Nut
                     IF ((bNutWeld_AlgNoNut_Active==TRUE) AND (bNutWeld_AlgNoNut_Step[10]==TRUE)) THEN
                        bNutWeld_AlgNoNut_Active=FALSE
                        bNutWeldAlgNoNutReq=FALSE
                        dopw_GunWork(nNutWeldGunNrSTK,FALSE)
                        dopw_NutIntensify(nNutWeldGunNrSTK,FALSE)
                        FOR nStepCnt=1 to 10
                           bNutWeld_AlgNoNut_Step[nStepCnt]=FALSE
                        ENDFOR
                        bNutWeld_TchAnlg_Active=FALSE
                        bNutWeldTchAnlgSTK=TRUE
                        $TIMER_STOP[nNutWeldManWeldTmr]=TRUE
                        $TIMER_STOP[nNutWeldSignalTmr]=TRUE
                        $TIMER[nNutWeldManWeldTmr]=-1000
                        $TIMER[nNutWeldSignalTmr]=-750
                        FOR nStepCnt=1 to 10
                           bNutWeld_TchAnlg_Step[nStepCnt]=FALSE
                        ENDFOR
                     ENDIF
                     IF ((bNutWeld_AlgNoNut_Active==TRUE) AND (bNutWeld_AlgNoNut_Step[6]==TRUE) AND (bNutWeld_AlgNoNut_Step[7]==FALSE)) THEN
                        bNutWeld_AlgNoNut_Active=FALSE
                        bNutWeldAlgNoNutReq=TRUE
                        FOR nStepCnt=1 to 10
                           bNutWeld_AlgNoNut_Step[nStepCnt]=FALSE
                        ENDFOR
                     ENDIF
                     IF ((bNutWeld_AlgNoNut_Active==TRUE) AND (bNutWeld_AlgNoNut_Step[5]==TRUE) AND (bNutWeld_AlgNoNut_Step[6]==FALSE)) THEN
                        IF (Exists_KrlDlg(nNutWeld_TA1Handle, nNutWeld_TA1Key)==FALSE) THEN
                           SWITCH nNutWeld_TA1Key
                              CASE 1 ; Accept - Store value and exit
                                 rNoNutValue[nNutWeldGunNrSTK]=rNutSensorValueTemp
                                 rNutSensorValueTemp=0.0
                                 bNutWeld_AlgNoNut_Step[10]=TRUE ; Reset Process
                              CASE 2 ; Rerun - discard value and re-execute
                                 rNutSensorValueTemp=0.0
                                 bNutWeld_AlgNoNut_Step[6]=TRUE ; Local Reset Process
                              CASE 3 ; Cancel - discard value and return to main selection
                                 rNutSensorValueTemp=0.0
                                 bNutWeld_AlgNoNut_Step[10]=TRUE ; Reset Process
                           ENDSWITCH
                        ENDIF
                        nNutWeld_TA1Key=0
                     ENDIF
                     IF ((bNutWeld_AlgNoNut_Active==TRUE) AND (bNutWeld_AlgNoNut_Step[4]==TRUE) AND (bNutWeld_AlgNoNut_Step[5]==FALSE)) THEN
                        rNutSensorValueTemp=ABS(aiNutSensor(nNutWeldGunNrSTK))
                        dopw_NutIntensify(nNutWeldGunNrSTK,FALSE)
                        dopw_GunWork(nNutWeldGunNrSTK,FALSE)
                        NutWeld_MsgPar[1]={par_type #value, par_real 0}
                        NutWeld_MsgPar[1].par_real=rNutSensorValueTemp
                        nNutWeld_TA1Handle = Set_KrlDlg (NutWeld_Msg[42], NutWeld_MsgPar[], NutWeld_SK_AcptRerun[], NutWeld_MsgOpt_NoStop)
                        bNutWeld_AlgNoNut_Step[5]=TRUE
                     ENDIF
                     IF ((bNutWeld_AlgNoNut_Active==TRUE) AND (bNutWeld_AlgNoNut_Step[3]==TRUE) AND (bNutWeld_AlgNoNut_Step[4]==FALSE)) THEN
                        ; Smart Electrode Dwell Time
                        IF ($TIMER_FLAG[nNutWeldManWeldTmr]==TRUE) THEN
                           $TIMER_STOP[nNutWeldSignalTmr]=TRUE
                           $TIMER[nNutWeldSignalTmr]=(-1000)
                           bNutWeld_AlgNoNut_Step[4]=TRUE
                        ENDIF
                     ENDIF
                     IF ((bNutWeld_AlgNoNut_Active==TRUE) AND (bNutWeld_AlgNoNut_Step[2]==TRUE) AND (bNutWeld_AlgNoNut_Step[3]==FALSE)) THEN
                        ; Check for Gun Closed
                        IF ($TIMER_FLAG[nNutWeldManWeldTmr]==TRUE) THEN
                           bNutWeld_AlgNoNut_Step[10]=TRUE ; Reset Process
                           nNutWeld_Handle_SPS=Set_Krlmsg (#NOTIFY, NutWeld_Msg[35], NutWeld_MsgPar[], NutWeld_MsgOpt_NoStop)
                        ELSE
                           IF (bpw_GunAtHome(nNutWeldGunNrSTK)==FALSE) THEN
                              $TIMER_STOP[nNutWeldSignalTmr]=TRUE
                              $TIMER[nNutWeldSignalTmr]=(-1000)
                              $TIMER_STOP[nNutWeldSignalTmr]=FALSE
                              bNutWeld_AlgNoNut_Step[3]=TRUE
                           ENDIF
                        ENDIF
                     ENDIF
                     IF ((bNutWeld_AlgNoNut_Active==TRUE) AND (bNutWeld_AlgNoNut_Step[1]==TRUE) AND (bNutWeld_AlgNoNut_Step[2]==FALSE)) THEN
                        IF (Exists_KrlDlg(nNutWeld_TA1Handle, nNutWeld_TA1Key)==FALSE) THEN
                           IF (nNutWeld_TA1Key==1) THEN
                              $TIMER_STOP[nNutWeldManWeldTmr]=FALSE
                              dopw_NutIntensify(nNutWeldGunNrSTK,FALSE)
                              dopw_GunWork(nNutWeldGunNrSTK,TRUE)
                              $TIMER_STOP[nNutWeldSignalTmr]=TRUE
                              $TIMER[nNutWeldSignalTmr]=(-750)
                              $TIMER_STOP[nNutWeldSignalTmr]=FALSE
                              bNutWeld_AlgNoNut_Step[2]=TRUE
                           ELSE
                              bNutWeld_AlgNoNut_Step[10]=TRUE ; Reset Process
                           ENDIF
                        ENDIF
                        nNutWeld_TA1Key=0
                     ENDIF
                     IF ((bNutWeldAlgNoNutReq==TRUE) AND (bNutWeld_AlgNoNut_Step[1]==FALSE)) THEN
                        bNutWeld_AlgNoNut_Active=TRUE
                        bNutWeld_AlgNoNut_Step[1]=TRUE
                        dopw_NutIntensify(nNutWeldGunNrSTK,FALSE)
                        dopw_GunWork(nNutWeldGunNrSTK,FALSE)
                        $TIMER_STOP[nNutWeldManWeldTmr]=TRUE
                        $TIMER[nNutWeldManWeldTmr]=(nNutWeld_ManWeld_Timeout*(-1000))
                        $TIMER_STOP[nNutWeldManWeldTmr]=FALSE
                        nNutWeld_TA1Key=0
                        nNutWeld_TA1Handle = Set_KrlDlg (NutWeld_Msg[40], NutWeld_MsgPar[], NutWeld_SK_CloseNWGun[], NutWeld_MsgOpt_NoStop)
                     ENDIF
                  ;ENDFOLD (USKB4-2.1 No Nut)
                  ;FOLD USKB4 Teach Selection
                     IF ((bNutWeld_TchAnlg_Active==TRUE) AND (bNutWeld_TchAnlg_Step[10]==TRUE)) THEN
                        bNutWeld_TchAnlg_Active=FALSE
                        bNutWeldTchAnlgSTK=FALSE
                        dopw_GunWork(nNutWeldGunNrSTK,FALSE)
                        dopw_NutIntensify(nNutWeldGunNrSTK,FALSE)
                        $TIMER_STOP[nNutWeldManWeldTmr]=TRUE
                        $TIMER_STOP[nNutWeldSignalTmr]=TRUE
                        $TIMER[nNutWeldManWeldTmr]=-1000
                        $TIMER[nNutWeldSignalTmr]=-750
                        FOR nStepCnt=1 to 10
                           bNutWeld_TchAnlg_Step[nStepCnt]=FALSE
                        ENDFOR
                     ENDIF
                     IF ((bNutWeld_TchAnlg_Active==TRUE) AND (bNutWeld_TchAnlg_Step[2]==TRUE) AND (bNutWeld_TchAnlg_Step[3]==FALSE)) THEN
                        IF (Exists_KrlDlg(nNutWeld_TAHandle, nNutWeld_TAKey)==FALSE) THEN
                           SWITCH nNutWeld_TAKey
                              CASE 1 ; No Nut
                                 bNutWeldAlgNoNutReq=TRUE
                                 bNutWeld_TchAnlg_Step[3]=TRUE
                              CASE 2 ; With Nut
                                 bNutWeldAlgWNutReq=TRUE
                                 bNutWeld_TchAnlg_Step[3]=TRUE
                              CASE 3 ; Invert Nut
                                 bNutWeldAlgInNutReq=TRUE
                                 bNutWeld_TchAnlg_Step[3]=TRUE
                              CASE 4 ; Check
                                 bNutWeldAlgCheckReq=TRUE
                                 bNutWeld_TchAnlg_Step[3]=TRUE
                              DEFAULT
                                 bNutWeld_TchAnlg_Step[3]=TRUE
                                 bNutWeld_TchAnlg_Step[10]=TRUE ; Reset Process
                           ENDSWITCH
                        ENDIF
                        nNutWeld_TAKey=0
                     ENDIF
                     IF ((bNutWeld_TchAnlg_Active==TRUE) AND (bNutWeld_TchAnlg_Step[1]==TRUE) AND (bNutWeld_TchAnlg_Step[2]==FALSE)) THEN
                        bNutWeld_TchAnlg_Step[2]=TRUE
                        nNutWeld_TAKey=0
                        NutWeld_MsgPar[1]={par_type #value, par_int 0}
                        NutWeld_MsgPar[1].par_int=nNutWeldGunNrSTK
                        nNutWeld_TAHandle = Set_KrlDlg (NutWeld_Msg[39], NutWeld_MsgPar[], NutWeld_SK_TchAnalog[], NutWeld_MsgOpt_NoStop)
                     ENDIF
                     IF ((bNutWeldTchAnlgSTK==TRUE) AND (bNutWeld_TchAnlg_Step[1]==FALSE)) THEN
                        bNutWeld_TchAnlg_Active=TRUE
                        bNutWeld_TchAnlg_Step[1]=TRUE
                     ENDIF
                  ;ENDFOLD (USKB4 Teach Selection)
               ;ENDFOLD (USKB4-4 Teach Analog)
               ;FOLD USKB4-4 Test Welding Current S225
                  IF ((bNutWeld_TstCrnt_Active==TRUE) AND (bNutWeld_TstCrnt_Step[10]==TRUE)) THEN
                     bNutWeld_TstCrnt_Active=FALSE
                     bNutWeldTstCrntSTK=FALSE
                     dopw_GunWork(nNutWeldGunNrSTK,FALSE)
                     dopw_WeldInit(nNutWeldGunNrSTK,FALSE)
                     dopw_NutIntensify(nNutWeldGunNrSTK,FALSE)
                     dopw_SetPrgNr(nNutWeldGunNrSTK, 0)
                     $TIMER_STOP[nNutWeldManWeldTmr]=TRUE
                     $TIMER_STOP[nNutWeldSignalTmr]=TRUE
                     $TIMER[nNutWeldManWeldTmr]=-1000
                     $TIMER[nNutWeldSignalTmr]=-750
                     FOR nStepCnt=1 to 10
                        bNutWeld_TstCrnt_Step[nStepCnt]=FALSE
                     ENDFOR
                  ENDIF
                  IF ((bNutWeld_TstCrnt_Active==TRUE) AND (bNutWeld_TstCrnt_Step[4]==TRUE) AND (bNutWeld_TstCrnt_Step[5]==FALSE)) THEN
                     ; Check for Weld Complete
                     IF ($TIMER_FLAG[nNutWeldManWeldTmr]==TRUE) THEN
                        bNutWeld_TstCrnt_Step[10]=TRUE ; Reset Process
                        nNutWeld_Handle_SPS=Set_Krlmsg (#NOTIFY, NutWeld_Msg[19], NutWeld_MsgPar[], NutWeld_MsgOpt_NoStop)
                     ELSE
                        IF (dipw_WeldComplete(nNutWeldGunNrSTK)==TRUE) THEN
                           dopw_WeldInit(nNutWeldGunNrSTK,FALSE)
                           dopw_NutIntensify(nNutWeldGunNrSTK,FALSE)
                           dopw_GunWork(nNutWeldGunNrSTK,FALSE)
                           bNutWeld_TstCrnt_Step[10]=TRUE
                           nNutWeld_Handle_SPS=Set_Krlmsg (#NOTIFY, NutWeld_Msg[45], NutWeld_MsgPar[], NutWeld_MsgOpt_NoStop)
                        ENDIF
                     ENDIF
                  ENDIF
                  IF ((bNutWeld_TstCrnt_Active==TRUE) AND (bNutWeld_TstCrnt_Step[3]==TRUE) AND (bNutWeld_TstCrnt_Step[4]==FALSE)) THEN
                     ; Check for Gun intensified
                     IF ($TIMER_FLAG[nNutWeldManWeldTmr]==TRUE) THEN
                        bNutWeld_TstCrnt_Step[10]=TRUE ; Reset Process
                        nNutWeld_Handle_SPS=Set_Krlmsg (#NOTIFY, NutWeld_Msg[18], NutWeld_MsgPar[], NutWeld_MsgOpt_NoStop)
                     ELSE
                        IF (dipw_IntensfPresOk(nNutWeldGunNrSTK)==TRUE) THEN
                           bNutWeld_TstCrnt_Step[4]=TRUE
                           dopw_SetPrgNr(nNutWeldGunNrSTK, nSpotNrTstCrnt )
                           ; Weld Initiate
                           dopw_WeldInit(nNutWeldGunNrSTK,TRUE)
                        ENDIF
                     ENDIF
                  ENDIF
                  IF ((bNutWeld_TstCrnt_Active==TRUE) AND (bNutWeld_TstCrnt_Step[2]==TRUE) AND (bNutWeld_TstCrnt_Step[3]==FALSE)) THEN
                     ; Check for Gun Closed
                     IF ($TIMER_FLAG[nNutWeldManWeldTmr]==TRUE) THEN
                        bNutWeld_TstCrnt_Step[10]=TRUE ; Reset Process
                        nNutWeld_Handle_SPS=Set_Krlmsg (#NOTIFY, NutWeld_Msg[35], NutWeld_MsgPar[], NutWeld_MsgOpt_NoStop)
                     ELSE
                        IF (($TIMER_FLAG[nNutWeldSignalTmr]==TRUE) AND (bpw_GunAtHome(nNutWeldGunNrSTK)==FALSE)) THEN
                           $TIMER_STOP[nNutWeldSignalTmr]=TRUE
                           $TIMER[nNutWeldSignalTmr]=(-500)
                           ; Intensify Gun
                           dopw_NutIntensify(nNutWeldGunNrSTK,TRUE)
                           bNutWeld_TstCrnt_Step[3]=TRUE
                        ENDIF
                     ENDIF
                  ENDIF
                  IF ((bNutWeld_TstCrnt_Active==TRUE) AND (bNutWeld_TstCrnt_Step[1]==TRUE) AND (bNutWeld_TstCrnt_Step[2]==FALSE)) THEN
                     IF (Exists_KrlDlg(nNutWeld_TCHandle, nNutWeld_TCKey)==FALSE) THEN
                        IF (nNutWeld_TCKey==1) THEN
                           $TIMER_STOP[nNutWeldManWeldTmr]=FALSE
                           dopw_NutIntensify(nNutWeldGunNrSTK,FALSE)
                           dopw_GunWork(nNutWeldGunNrSTK,TRUE)
                           $TIMER_STOP[nNutWeldSignalTmr]=TRUE
                           $TIMER[nNutWeldSignalTmr]=(-750)
                           $TIMER_STOP[nNutWeldSignalTmr]=FALSE
                           bNutWeld_TstCrnt_Step[2]=TRUE
                        ELSE
                           bNutWeld_TstCrnt_Step[10]=TRUE ; Reset Process
                        ENDIF
                     ENDIF
                     nNutWeld_TCKey=0
                  ENDIF
                  IF ((bNutWeldTstCrntSTK==TRUE) AND (bNutWeld_TstCrnt_Step[1]==FALSE)) THEN
                     IF (bNutWeldWOJoining==FALSE) THEN
                        bNutWeld_TstCrnt_Active=TRUE
                        bNutWeld_TstCrnt_Step[1]=TRUE
                        $TIMER_STOP[nNutWeldManWeldTmr]=TRUE
                        $TIMER[nNutWeldManWeldTmr]=(nNutWeld_ManWeld_Timeout*(-1000))
                        nNutWeld_TCKey=0
                        NutWeld_MsgPar[1]={par_type #value, par_int 0}
                        NutWeld_MsgPar[1].par_int=nNutWeldGunNrSTK
                        nNutWeld_TCHandle = Set_KrlDlg (NutWeld_Msg[36], NutWeld_MsgPar[], NutWeld_SK_TstCncl[], NutWeld_MsgOpt_NoStop)
                     ELSE
                        nNutWeld_Handle_SPS=Set_Krlmsg (#NOTIFY, NutWeld_Msg[33], NutWeld_MsgPar[], NutWeld_MsgOpt_NoStop)
                        bNutWeldTstCrntSTK=FALSE
                     ENDIF
                  ENDIF
               ;ENDFOLD (USKB4-4 Test Welding Current S225)
            ;ENDFOLD (USKB4 - Gun Maintenance Actions)
         ;ENDFOLD (Status Key Control)
         ;FOLD Status Hopper Low Level
            ;FOLD Hopper1 Low Level
               ; No warning turn on Green light
               IF (dipw1_HopperLowLevel==TRUE) THEN
                  dopw1_LevelOk=TRUE
                  dopw1_LowLevel=FALSE
               ELSE
                  ; warning Off on Red light
                  IF (dipw1_HopperLowLevel==FALSE) THEN
                     dopw1_LevelOk=FALSE
                     dopw1_LowLevel=TRUE
                  ENDIF
               ENDIF
            ;ENDFOLD (Hopper1 Low Level)
            ;FOLD Hopper2 Low Level
               ; No warning turn on Green light
               IF (dipw2_HopperLowLevel==TRUE) THEN
                  dopw2_LevelOk=TRUE
                  dopw2_LowLevel=FALSE
               ELSE
                  ; warning Off on Red light
                  IF (dipw2_HopperLowLevel==FALSE) THEN
                     dopw2_LevelOk=FALSE
                     dopw2_LowLevel=TRUE
                  ENDIF
               ENDIF
            ;ENDFOLD (Hopper2 Low Level)
            ;FOLD Hopper3 Low Level
               ; No warning turn on Green light
               IF (dipw3_HopperLowLevel==TRUE) THEN
                  dopw3_LevelOk=TRUE
                  dopw3_LowLevel=FALSE
               ELSE
                  ; warning Off on Red light
                  IF (dipw3_HopperLowLevel==FALSE) THEN
                     dopw3_LevelOk=FALSE
                     dopw3_LowLevel=TRUE
                  ENDIF
               ENDIF
            ;ENDFOLD (Hopper3 Low Level)
         ;ENDFOLD (Status Hopper Low Level)
         ;FOLD Status Stepper warning EOL
            ;FOLD Stepper warning Gun1
               ; No warning or end of electrode life turn on Green light
               IF ((dipw1_StepperWarning==FALSE) AND (dipw1_EndOfStepper==FALSE)) THEN
                  dopw1_StepperWarningPL=TRUE
                  dopw1_EndofStepperPL=FALSE
                  ; Warning Only no end of electrode life turn on Amber light
               ELSE
                  IF ((dipw1_StepperWarning==TRUE) AND (dipw1_EndOfStepper==FALSE)) THEN
                     dopw1_StepperWarningPL=TRUE
                     dopw1_EndofStepperPL=TRUE
                     ; warning Off  Electrode at end of life turn on Red light
                  ELSE
                     IF (dipw1_EndOfStepper==TRUE) THEN
                        dopw1_StepperWarningPL=FALSE
                        dopw1_EndofStepperPL=TRUE
                     ENDIF
                  ENDIF
               ENDIF
            ;ENDFOLD Stepper warning Gun1
            ;FOLD Stepper warning Gun2
               ; No warning or end of electrode life turn on Green light
               IF ((dipw2_StepperWarning==FALSE) AND (dipw2_EndOfStepper==FALSE)) THEN
                  dopw2_StepperWarningPL=TRUE
                  dopw2_EndofStepperPL=FALSE
                  ; Warning Only no end of electrode life turn on Amber light
               ELSE
                  IF ((dipw2_StepperWarning==TRUE) AND (dipw2_EndOfStepper==FALSE)) THEN
                     dopw2_StepperWarningPL=TRUE
                     dopw2_EndofStepperPL=TRUE
                     ; warning Off  Electrode at end of life turn on Red light
                  ELSE
                     IF (dipw2_EndOfStepper==TRUE) THEN
                        dopw2_StepperWarningPL=FALSE
                        dopw2_EndofStepperPL=TRUE
                     ENDIF
                  ENDIF
               ENDIF
            ;ENDFOLD Stepper warning Gun2
            ;FOLD Stepper warning Gun3
               ; No warning or end of electrode life turn on Green light
               IF ((dipw3_StepperWarning==FALSE) AND (dipw3_EndOfStepper==FALSE)) THEN
                  dopw3_StepperWarningPL=TRUE
                  dopw3_EndofStepperPL=FALSE
                  ; Warning Only no end of electrode life turn on Amber light
               ELSE
                  IF ((dipw3_StepperWarning==TRUE) AND (dipw3_EndOfStepper==FALSE)) THEN
                     dopw3_StepperWarningPL=TRUE
                     dopw3_EndofStepperPL=TRUE
                     ; warning Off  Electrode at end of life turn on Red light
                  ELSE
                     IF (dipw3_EndOfStepper==TRUE) THEN
                        dopw3_StepperWarningPL=FALSE
                        dopw3_EndofStepperPL=TRUE
                     ENDIF
                  ENDIF
               ENDIF
            ;ENDFOLD Stepper warning Gun3
         ;ENDFOLD (Status Stepper warning EOL)
      ;ENDFOLD (Implementation)
   ;ENDFOLD (Details)
   rNutSensorValue[1] = aiNutSensorPW1
   rNutSensorValue[2] = aiNutSensorPW2
   rNutSensorValue[3] = aiNutSensorPW3
   rStrokeSensorValue[1] = aipw1_LVDT
   rStrokeSensorValue[2] = aipw2_LVDT
   rStrokeSensorValue[3] = aipw3_LVDT
   bpw1_GunAtHome = (aipw1_LVDT < (raipw1_LVDT_OPN + 350)) AND (aipw1_LVDT > (raipw1_LVDT_OPN - 350))
   bpw2_GunAtHome = (aipw2_LVDT < (raipw2_LVDT_OPN + 250)) AND (aipw2_LVDT > (raipw2_LVDT_OPN - 250))
   bpw3_GunAtHome = (aipw3_LVDT < (raipw3_LVDT_OPN + 100)) AND (aipw3_LVDT > (raipw3_LVDT_OPN - 100))
   bpw1_GunAtWork = (aipw1_LVDT < (raipw1_LVDT_CLS_W_NUT + 150)) AND (aipw1_LVDT > (raipw1_LVDT_CLS_W_NUT - 150))
   bpw2_GunAtWork = (aipw2_LVDT < (raipw2_LVDT_CLS_W_NUT + 150)) AND (aipw2_LVDT > (raipw2_LVDT_CLS_W_NUT - 150))
   bpw3_GunAtWork = (aipw3_LVDT < (raipw3_LVDT_CLS_W_NUT + 100)) AND (aipw3_LVDT > (raipw3_LVDT_CLS_W_NUT - 100))
   IF ((iLastActiveGun==1) OR (iLastActiveGun==2) OR (iLastActiveGun==3)) THEN
      rLowerLVDT=rNutSensorValue[iLastActiveGun]
      rUpperLVDT=rStrokeSensorValue[iLastActiveGun]
   ELSE
      rLowerLVDT=0
      rUpperLVDT=0
   ENDIF

   bDumpNutExceeded=NOT (nDumpNutRetries <= nMaxDumpNutRetries)
END ; (NutWeld_Bkg)

GLOBAL DEF NutWeld_PreWeld (nutweldINFO :IN)
   ;FOLD Details
      ;FOLD Declaration
         DECL NutWeldDAT nutweldINFO
      ;ENDFOLD (Declaration)
      ;FOLD Implementation
         PWInitUserIO(nutweldINFO)
         PreNutWeldSup(nutweldINFO)
         dopw_SetPrgNr(nutweldINFO.GunNr, nutweldINFO.SpotNr )
         IF (bNutWeld_PreAdvPin==TRUE) THEN
            dopw_PinAdv(nutweldINFO.GunNr, TRUE)
         ENDIF
         bNutWeld_PreWeld_Cmplt=TRUE
      ;ENDFOLD (Implementation)
   ;ENDFOLD (Details)
END ; (NutWeld_PreWeld)

GLOBAL DEF NutWeld_Weld(nutweldINFO :IN,WeldPos:IN, WeldBase:IN, EnableReload:IN, Move1:IN, Move2:IN, Move3:IN, ReloadPos1:IN, ReloadPos2:IN, ReloadPos3:IN, ReloadBase1:IN, ReloadBase2:IN, ReloadBase3:IN)
   ;FOLD Details
      ;FOLD Declaration
         INT EnableReload
         E6POS WeldPos,ReloadPos1,ReloadPos2,ReloadPos3
         DECL FDAT WeldBase,ReloadBase1,ReloadBase2,ReloadBase3
         DECL Nut_Dump_Move Move1,Move2,Move3
         DECL NutWeldDAT nutweldINFO
      ;ENDFOLD (Declaration)
      ;FOLD Implementation
         ;If no Reloadpos is specified, the variable must be set to default values
         EnableReload=3
         SWITCH (EnableReload)
            CASE 0
               Move1=#Reload_PTP
               ReloadPos1=WeldPos
               ReloadBase1=WeldBase
               Move2=#Reload_PTP
               ReloadPos2=WeldPos
               ReloadBase2=WeldBase
               Move3=#Reload_PTP
               ReloadPos3=WeldPos
               ReloadBase3=WeldBase
            CASE 1
               Move2=#Reload_PTP
               ReloadPos2=WeldPos
               ReloadBase2=WeldBase
               Move3=#Reload_PTP
               ReloadPos3=WeldPos
               ReloadBase3=WeldBase
            CASE 2
               Move3=#Reload_PTP
               ReloadPos3=WeldPos
               ReloadBase3=WeldBase
            CASE 3
         ENDSWITCH
         WAIT FOR (nDumpNutRetries <= nMaxDumpNutRetries)
         WAIT FOR (bNutWeld_PreWeld_Cmplt==TRUE)
         bDump_Nut=FALSE
         eCurrentState=#FeedRequest
         FeedNutReq(nutweldINFO)
         eCurrentState=#CloseGun
         CloseNutGun(nutweldINFO)
         IF (bDump_Nut == TRUE) THEN
            ; do nothing here
         ELSE
            IF NOT (eCurrentState==#ERRORCloseGun) THEN
               eCurrentState=#CheckNut
            ENDIF
            CheckNutPresent(nutweldINFO)
            IF (bDump_Nut == TRUE) THEN
               IF NOT (eCurrentState==#ERRORCloseGun) THEN
                  IF NOT (eCurrentState==#ERRORInvertedNut) THEN
                     IF NOT (eCurrentState==#ERRORNoNut) THEN
                        eCurrentState=#DumpNut
                     ENDIF
                  ENDIF
               ENDIF
               ; do nothing here
            ENDIF
         ENDIF

         bNutFeedOK=NOT bDump_Nut
         IF ((bDump_Nut == TRUE) AND (nDumpNutRetries <= nMaxDumpNutRetries)) THEN
            nDumpNutRetries=nDumpNutRetries+1
            bDump_Nut=FALSE
            IF NOT (eCurrentState==#ERRORCloseGun) THEN
               IF NOT (eCurrentState==#ERRORInvertedNut) THEN
                  IF NOT (eCurrentState==#ERRORNoNut) THEN
                     eCurrentState=#OpenGun
                  ENDIF
               ENDIF
            ENDIF
            OpenNutGun(nutweldINFO)
         ELSE
            eCurrentState=#IntensifyGun
            IntensfNutGun(nutweldINFO)
            IF (PNWStyle==#STUDWELD) THEN
               dopw_PinAdv(nutweldINFO.GunNr, FALSE)
            ENDIF
            IF NOT (eCurrentState==#ERRORCloseGun) THEN
               IF NOT (eCurrentState==#ERRORInvertedNut) THEN
                  IF NOT (eCurrentState==#ERRORNoNut) THEN
                     IF NOT (eCurrentState==#ERRORIntensifyWelder) THEN
                        eCurrentState=#WeldInitiate
                     ENDIF
                  ENDIF
               ENDIF
            ENDIF
            WeldInitiate(nutweldINFO)
            IF (bElectChangeReq==TRUE) THEN
               nElectChangeReq=nElectChangeReq+1
            ENDIF
            dopw_PinAdv(nutweldINFO.GunNr, FALSE)
            IF NOT (eCurrentState==#ERRORCloseGun) THEN
               IF NOT (eCurrentState==#ERRORInvertedNut) THEN
                  IF NOT (eCurrentState==#ERRORNoNut) THEN
                     IF NOT (eCurrentState==#ERRORIntensifyWelder) THEN
                        eCurrentState=#OpenGun
                     ENDIF
                  ENDIF
               ENDIF
            ENDIF
            OpenNutGun(nutweldINFO)
            IF ((dipw_EndOfStepper(nutweldINFO.GunNr)==TRUE) OR (dipw_StepperWarning(nutweldINFO.GunNr)==TRUE)) THEN
               SWITCH nutweldINFO.GunNr
                  CASE 1
                     bElectrodeAtEOL_1 = TRUE;
                  CASE 2
                     bElectrodeAtEOL_2 = TRUE;
                  CASE 3
                     bElectrodeAtEOL_3 = TRUE;
               ENDSWITCH
            ENDIF
            dopw_SetPrgNr(nutweldINFO.GunNr, 0 )
            IF (bNutWeld_PreAdvPin==TRUE) THEN
               dopw_PinAdv(nutweldINFO.GunNr, TRUE)
            ENDIF
            nDumpNutRetries=0
            bDump_Nut=FALSE
         ENDIF
         WAIT FOR (((bpw_GunAtHome(nutweldINFO.GunNr)==TRUE) AND (bpw_GunAtWork(nutweldINFO.GunNr)==FALSE)))

         IF NOT (eCurrentState==#ERRORCloseGun) THEN
            IF NOT (eCurrentState==#ERRORInvertedNut) THEN
               IF NOT (eCurrentState==#ERRORNoNut) THEN
                  IF NOT (eCurrentState==#ERRORIntensifyWelder) THEN
                     eCurrentState=#GunHome
                  ENDIF
               ENDIF
            ENDIF
         ENDIF
      ;ENDFOLD (Implementation)
   ;ENDFOLD (Details)
END ; (NutWeld_Weld)

DEF NutWeld_ProcessReset( )
   ;FOLD Details
      ;FOLD Declaration
      ;ENDFOLD (Declaration)
      ;FOLD Implementation
         bNutWeld_PreWeld_Cmplt=FALSE
         dopw_SetPrgNr(1, 0)
         dopw_SetPrgNr(2, 0)
         dopw_SetPrgNr(3, 0)
         dopw_WeldInit(1,FALSE)
         dopw_WeldInit(2,FALSE)
         dopw_WeldInit(3,FALSE)
         dopw_NutIntensify(1,FALSE)
         dopw_NutIntensify(2,FALSE)
         dopw_NutIntensify(3,FALSE)
         dopw_BlowOff(1,FALSE)
         dopw_BlowOff(2,FALSE)
         dopw_BlowOff(3,FALSE)
      ;ENDFOLD (Implementation)
   ;ENDFOLD (Details)
END ; (NutWeld_ProcessReset)

DEF PWInitUserIO(nutweldINFO :IN )
   ;FOLD Details
      ;FOLD Declaration
         DECL NutWeldDAT nutweldINFO
      ;ENDFOLD (Declaration)
      ;FOLD Implementation


         ;DECL GLOBAL REAL rLowTol[3] lower LVDT
         rLowTol[1]=rSetLowerLVDT_CLS_W_NUT[1]-250
         rLowTol[2]=rSetLowerLVDT_CLS_W_NUT[2]-600
         rLowTol[3]=rSetLowerLVDT_CLS_W_NUT[3]-850
         ;DECL GLOBAL REAL rHighTol[3] lower LVDT
         rHighTol[1]=rSetLowerLVDT_CLS_W_NUT[1]+250
         rHighTol[2]=rSetLowerLVDT_CLS_W_NUT[2]+600
         rHighTol[3]=rSetLowerLVDT_CLS_W_NUT[3]+850

         ;DECL GLOBAL REAL rLowLVDT[3] upper LVDT
         rLowLVDT[1]=rSetUpperLVDT_CLS_W_NUT[1]-150
         rLowLVDT[2]=rSetUpperLVDT_CLS_W_NUT[2]-150
         rLowLVDT[3]=rSetUpperLVDT_CLS_W_NUT[3]-300
         ;DECL GLOBAL REAL rHighLVDT[3] upper LVDT
         rHighLVDT[1]=rSetUpperLVDT_CLS_W_NUT[1]+150
         rHighLVDT[2]=rSetUpperLVDT_CLS_W_NUT[2]+150
         rHighLVDT[3]=rSetUpperLVDT_CLS_W_NUT[3]+100
         raipw1_LVDT_CLS_W_NUT=rSetUpperLVDT_CLS_W_NUT[1]
         raipw2_LVDT_CLS_W_NUT=rSetUpperLVDT_CLS_W_NUT[2]
         raipw3_LVDT_CLS_W_NUT=rSetUpperLVDT_CLS_W_NUT[3]

         iLastActiveGun=nutweldINFO.GunNr
         rNutSensorValueInUse=rNutSensorValue[nutweldINFO.GunNr]
         rStrokeSensorValueInUse=rStrokeSensorValue[nutweldINFO.GunNr]
         rNutInvertedValueInUse=rNutInvertedValue[nutweldINFO.GunNr]
         rNoNutValueInUse=rNoNutValue[nutweldINFO.GunNr]
         rNutPresentValueInUse=rNutPresentValue[nutweldINFO.GunNr]
         rNutSensorTolInUse=rNutSensorTolerance[nutweldINFO.GunNr]
         rNutSensorTol2InUse=rNutSensorTolerance2[nutweldINFO.GunNr]
         rLowTolInUse=rLowTol[nutweldINFO.GunNr]
         rHighTolInUse=rHighTol[nutweldINFO.GunNr]
         rLowLVDTTolInUse=rLowLVDT[nutweldINFO.GunNr]
         rHighLVDTTolInUse=rHighLVDT[nutweldINFO.GunNr]
      ;ENDFOLD (Implementation)
   ;ENDFOLD (Details)
END ; (PWInitUserIO)

DEF PreNutWeldSup(nutweldINFO :IN )
   ;FOLD Details
      ;FOLD Declaration
         DECL NutWeldDAT nutweldINFO
         BOOL bMsgRelease
         BOOL bSkipTempChk
         BOOL bSkipWtrChk
         BOOL bSkipWtrTempChk
         BOOL bSkipPressSwChk
         BOOL bSkipTimerRdy
         BOOL bSkipWeldFault
         BOOL bSkipFdrHmChk
         BOOL bSkipPinRetChk
      ;ENDFOLD (Declaration)
      ;FOLD Implementation
         bMsgRelease=FALSE
         bSkipTempChk=FALSE
         bSkipWtrChk=FALSE
         bSkipWtrTempChk=FALSE
         bSkipPressSwChk=FALSE
         bSkipTimerRdy=FALSE
         bSkipWeldFault=FALSE
         bSkipFdrHmChk=FALSE
         bSkipPinRetChk=FALSE
         bGunReady2Start=FALSE
         iSpotnr=nutweldINFO.SpotNr
         eCurrentState=#GunHome
         ; Reset Outputs
         dopw_StartFeed(nutweldINFO.GunNr,FALSE)
         dopw_WeldInit(nutweldINFO.GunNr,FALSE)
         dopw1_FaultReset=TRUE
         dopw2_FaultReset=TRUE
         dopw3_FaultReset=TRUE
         nFeedRetries=0
         nWeldRetries=0
         OpenNutGun(nutweldINFO) ; Open Gun
         ;FOLD Check the Tranformer Temperature Switch
            WAIT FOR dipw_XtfmrTempOk(nutweldINFO.GunNr)
            WAIT FOR NOT bSkipTempChk
            WHILE ((bNutWeldWOJoining==FALSE) AND (dipw_XtfmrTempOk(nutweldINFO.GunNr)==FALSE) AND (bSkipTempChk==FALSE))
               ;FOLD Dialog "Nut Welder Over Temp Fault!  Transformer Switch Is Not On!"
                  REPEAT
                     nNutWeld_Handle = Set_KrlDlg (NutWeld_Msg[4], NutWeld_MsgPar[], NutWeld_SK_RetrySkip[], NutWeld_MsgOpt_Stop)
                     IF (nNutWeld_Handle > 0) THEN
                        WHILE (Exists_KrlDlg(nNutWeld_Handle, nNutWeld_Key))
                           IF ($ERR.Int_Prio>0) THEN
                              BRAKE
                           ENDIF
                           WAIT SEC 0.024
                        ENDWHILE
                        SWITCH nNutWeld_Key
                           CASE 1 ; Diagnostic
                              nNutWeld_Handle = Set_Krlmsg (#QUIT, NutWeld_Msg[2], NutWeld_MsgPar[], NutWeld_MsgOpt_Stop)
                              WHILE (Exists_KrlMsg(nNutWeld_Handle))
                                 WAIT SEC 0.024
                              ENDWHILE
                           CASE 2 ; Retry
                              WAIT SEC 0.100
                              bMsgRelease=TRUE
                           CASE 3 ; Skip
                              WAIT SEC 0.100
                              bMsgRelease=TRUE
                              bSkipTempChk=TRUE
                        ENDSWITCH
                     ENDIF
                  UNTIL (bMsgRelease==TRUE)
                  bMsgRelease=FALSE
               ;ENDFOLD (Dialog)
            ENDWHILE
         ;ENDFOLD (Check the Tranformer Temperature Switch)
         bGunReady2Start=NOT bNutWeldWOJoining AND dipw_XtfmrTempOk(nutweldINFO.GunNr) AND NOT bSkipTempChk
         ;FOLD Check the Water is Flowing
            WAIT FOR dipw_WaterOk(nutweldINFO.GunNr)
            WAIT FOR NOT bSkipWtrChk
            WHILE ((bNutWeldWOJoining==FALSE) AND (dipw_WaterOk(nutweldINFO.GunNr)==FALSE) AND (bSkipWtrChk==FALSE))
               ;FOLD Dialog "Nut Welder Water Flow Fault!  Water Flow Switch Is Not On!"
                  REPEAT
                     nNutWeld_Handle = Set_KrlDlg (NutWeld_Msg[5], NutWeld_MsgPar[], NutWeld_SK_StrtWtrSkip[], NutWeld_MsgOpt_Stop)
                     IF (nNutWeld_Handle > 0) THEN
                        WHILE (Exists_KrlDlg(nNutWeld_Handle, nNutWeld_Key))
                           IF ($ERR.Int_Prio>0) THEN
                              BRAKE
                           ENDIF
                           WAIT SEC 0.024
                        ENDWHILE
                        SWITCH nNutWeld_Key
                           CASE 1 ; Diagnostic
                              nNutWeld_Handle = Set_Krlmsg (#QUIT, NutWeld_Msg[2], NutWeld_MsgPar[], NutWeld_MsgOpt_Stop)
                              WHILE (Exists_KrlMsg(nNutWeld_Handle))
                                 WAIT SEC 0.024
                              ENDWHILE
                           CASE 2 ; Start Water
                              dopw_StartWater(nutweldINFO.GunNr,TRUE)
                              nNutWeld_Handle=Set_Krlmsg (#STATE, NutWeld_Msg[6], NutWeld_MsgPar[], NutWeld_MsgOpt_NoStop)
                              WAIT SEC nNutWeld_WtrStrtTime ; (Default:  4)
                              bNutWeld_Clear=Clear_KRLMsg(nNutWeld_Handle)
                              bMsgRelease=TRUE
                           CASE 3 ; Skip
                              WAIT SEC 0.100
                              bMsgRelease=TRUE
                              bSkipWtrChk=TRUE
                        ENDSWITCH
                     ENDIF
                  UNTIL (bMsgRelease==TRUE)
                  bMsgRelease=FALSE
               ;ENDFOLD (Dialog)
            ENDWHILE
         ;ENDFOLD (Check the Water is Flowing)
         bGunReady2Start=bGunReady2Start AND dipw_WaterOk(nutweldINFO.GunNr) AND NOT bSkipWtrChk
         ;FOLD Check the Temperature Water
            WAIT FOR dipw_WaterTempOk(nutweldINFO.GunNr)
            WAIT FOR NOT bSkipWtrTempChk
            WHILE ((bNutWeldWOJoining==FALSE) AND (dipw_WaterTempOk(nutweldINFO.GunNr)==FALSE) AND (bSkipWtrTempChk==FALSE))
               IF NOT di472WaterTempOK THEN
                  $LOOP_MSG[] = " No WaterTemp in Gun1                                                                                                  "
               ENDIF
               IF NOT di520WaterTempOK THEN
                  $LOOP_MSG[] = " No WaterTemp in Gun2                                                                                                  "
               ENDIF
               IF NOT di568WaterTempOK THEN
                  $LOOP_MSG[] = " No WaterTemp in Gun3                                                                                                  "
               ENDIF
            ENDWHILE
            $LOOP_MSG[] = "                                                                                                                    "
         ;ENDFOLD (Check the Temperature Water)
         bGunReady2Start=bGunReady2Start AND dipw_WaterTempOk(nutweldINFO.GunNr)
         ;FOLD Check that the Pressure Switch is off
            WAIT FOR NOT dipw_IntensfPresOk(nutweldINFO.GunNr)
            WAIT FOR NOT bSkipPressSwChk
            WHILE ((bNutWeldWOJoining==FALSE) AND (dipw_IntensfPresOk(nutweldINFO.GunNr)==TRUE) AND (bSkipPressSwChk==FALSE))
               ;FOLD Dialog "Nut Welder Intensify Pressure Fault!  Pressure Switch Is Not Off!"
                  REPEAT
                     nNutWeld_Handle = Set_KrlDlg (NutWeld_Msg[7], NutWeld_MsgPar[], NutWeld_SK_RetrySkip[], NutWeld_MsgOpt_Stop)
                     IF (nNutWeld_Handle > 0) THEN
                        WHILE (Exists_KrlDlg(nNutWeld_Handle, nNutWeld_Key))
                           IF ($ERR.Int_Prio>0) THEN
                              BRAKE
                           ENDIF
                           WAIT SEC 0.024
                        ENDWHILE
                        SWITCH nNutWeld_Key
                           CASE 1 ; Diagnostic
                              nNutWeld_Handle = Set_Krlmsg (#QUIT, NutWeld_Msg[2], NutWeld_MsgPar[], NutWeld_MsgOpt_Stop)
                              WHILE (Exists_KrlMsg(nNutWeld_Handle))
                                 WAIT SEC 0.024
                              ENDWHILE
                           CASE 2 ; Retry
                              WAIT SEC 0.100
                              bMsgRelease=TRUE
                           CASE 3 ; Skip
                              WAIT SEC 0.100
                              bMsgRelease=TRUE
                              bSkipPressSwChk=TRUE
                        ENDSWITCH
                     ENDIF
                  UNTIL (bMsgRelease==TRUE)
                  bMsgRelease=FALSE
               ;ENDFOLD (Dialog)
            ENDWHILE
         ;ENDFOLD (Check that the Pressure Switch is off)
         bGunReady2Start=bGunReady2Start AND NOT dipw_IntensfPresOk(nutweldINFO.GunNr) AND NOT bSkipPressSwChk
         ;FOLD Check that the Timer Is Ready To Weld
            WAIT FOR dipw_Ready(nutweldINFO.GunNr)
            WAIT FOR NOT bSkipTimerRdy
            WHILE ((bNutWeldWOJoining==FALSE) AND (dipw_Ready(nutweldINFO.GunNr)==FALSE) AND (bSkipTimerRdy==FALSE))
               ;FOLD Dialog "Bosch Timer Not Ready Fault!!!"
                  REPEAT
                     nNutWeld_Handle = Set_KrlDlg (NutWeld_Msg[8], NutWeld_MsgPar[], NutWeld_SK_ResetSkip[], NutWeld_MsgOpt_Stop)
                     IF (nNutWeld_Handle > 0) THEN
                        WHILE (Exists_KrlDlg(nNutWeld_Handle, nNutWeld_Key))
                           IF ($ERR.Int_Prio>0) THEN
                              BRAKE
                           ENDIF
                           WAIT SEC 0.024
                        ENDWHILE
                        SWITCH nNutWeld_Key
                           CASE 1 ; Diagnostic
                              nNutWeld_Handle = Set_Krlmsg (#QUIT, NutWeld_Msg[2], NutWeld_MsgPar[], NutWeld_MsgOpt_Stop)
                              WHILE (Exists_KrlMsg(nNutWeld_Handle))
                                 WAIT SEC 0.024
                              ENDWHILE
                           CASE 2 ; Reset
                              dopw_FaultReset(nutweldINFO.GunNr,FALSE)
                              WAIT SEC 0.050
                              dopw_FaultReset(nutweldINFO.GunNr,TRUE)
                              WAIT SEC 0.5
                              dopw_FaultReset(nutweldINFO.GunNr,FALSE)
                              bMsgRelease=TRUE
                           CASE 3 ; Skip
                              WAIT SEC 0.100
                              bMsgRelease=TRUE
                              bSkipTimerRdy=TRUE
                        ENDSWITCH
                     ENDIF
                  UNTIL (bMsgRelease==TRUE)
                  bMsgRelease=FALSE
               ;ENDFOLD (Dialog)
            ENDWHILE
         ;ENDFOLD (Check that the Timer Is Ready To Weld)
         bGunReady2Start=bGunReady2Start AND dipw_Ready(nutweldINFO.GunNr) AND NOT bSkipTimerRdy
         ;FOLD Check that the Timer Has No Faults
            dopw1_FaultReset=FALSE
            dopw2_FaultReset=FALSE
            dopw3_FaultReset=FALSE
            WAIT FOR NOT dipw_Fault(nutweldINFO.GunNr)
            WAIT FOR NOT bSkipWeldFault
            WHILE ((bNutWeldWOJoining==FALSE) AND (dipw_Fault(nutweldINFO.GunNr)==TRUE) AND (bSkipWeldFault==FALSE))
               dopw_FaultReset(nutweldINFO.GunNr,TRUE)
               WAIT SEC 0.5
               dopw_FaultReset(nutweldINFO.GunNr,FALSE)
               $TIMER_STOP[nNutWeldSignalTmr]=TRUE
               $TIMER[nNutWeldSignalTmr]=nNutWeld_Signal_Timeout*(-1)
               $TIMER_STOP[nNutWeldSignalTmr]=FALSE
               WAIT FOR ((dipw_Fault(nutweldINFO.GunNr)==FALSE) OR ($TIMER_FLAG[nNutWeldSignalTmr]==TRUE))
               $TIMER_STOP[nNutWeldSignalTmr]=TRUE
               ;FOLD Dialog "Weld Timer has a Weld Fault!!!"
                  IF ((bNutWeldWOJoining==FALSE) AND (dipw_Fault(nutweldINFO.GunNr)==TRUE) AND (bSkipWeldFault==FALSE)) THEN
                     REPEAT
                        nNutWeld_Handle = Set_KrlDlg (NutWeld_Msg[9], NutWeld_MsgPar[], NutWeld_SK_ResetSkip[], NutWeld_MsgOpt_Stop)
                        IF (nNutWeld_Handle > 0) THEN
                           WHILE (Exists_KrlDlg(nNutWeld_Handle, nNutWeld_Key))
                              IF ($ERR.Int_Prio>0) THEN
                                 BRAKE
                              ENDIF
                              WAIT SEC 0.024
                           ENDWHILE
                           SWITCH nNutWeld_Key
                              CASE 1 ; Diagnostic
                                 nNutWeld_Handle = Set_Krlmsg (#QUIT, NutWeld_Msg[2], NutWeld_MsgPar[], NutWeld_MsgOpt_Stop)
                                 WHILE (Exists_KrlMsg(nNutWeld_Handle))
                                    WAIT SEC 0.024
                                 ENDWHILE
                              CASE 2 ; Reset
                                 bMsgRelease=TRUE
                              CASE 3 ; Skip
                                 WAIT SEC 0.100
                                 bMsgRelease=TRUE
                                 bSkipWeldFault=TRUE
                           ENDSWITCH
                        ENDIF
                     UNTIL (bMsgRelease==TRUE)
                  ENDIF
                  bMsgRelease=FALSE
               ;ENDFOLD (Dialog)
            ENDWHILE
         ;ENDFOLD (Check that the Timer Has No Faults)
         bGunReady2Start=bGunReady2Start AND NOT dipw_Fault(nutweldINFO.GunNr) AND NOT bSkipWeldFault
         ;FOLD Check that the Nut Feeder is Home
            WAIT FOR dipw_SpearHome(nutweldINFO.GunNr)
            WAIT FOR NOT bSkipFdrHmChk
            WHILE ((bNutWeldWOJoining==FALSE) AND (dipw_SpearHome(nutweldINFO.GunNr)==FALSE) AND (bSkipFdrHmChk==FALSE))
               ;FOLD Dialog "Nut Feeder is Not Home Fault!"
                  REPEAT
                     nNutWeld_Handle = Set_KrlDlg (NutWeld_Msg[47], NutWeld_MsgPar[], NutWeld_SK_RetrySkip[], NutWeld_MsgOpt_Stop)
                     IF (nNutWeld_Handle > 0) THEN
                        WHILE (Exists_KrlDlg(nNutWeld_Handle, nNutWeld_Key))
                           IF ($ERR.Int_Prio>0) THEN
                              BRAKE
                           ENDIF
                           WAIT SEC 0.024
                        ENDWHILE
                        SWITCH nNutWeld_Key
                           CASE 1 ; Diagnostic
                              nNutWeld_Handle = Set_Krlmsg (#QUIT, NutWeld_Msg[2], NutWeld_MsgPar[], NutWeld_MsgOpt_Stop)
                              WHILE (Exists_KrlMsg(nNutWeld_Handle))
                                 WAIT SEC 0.024
                              ENDWHILE
                           CASE 2 ; Retry
                              WAIT SEC 0.100
                              bMsgRelease=TRUE
                           CASE 3 ; Skip
                              WAIT SEC 0.100
                              bMsgRelease=TRUE
                              bSkipFdrHmChk=TRUE
                        ENDSWITCH
                     ENDIF
                  UNTIL (bMsgRelease==TRUE)
                  bMsgRelease=FALSE
               ;ENDFOLD (Dialog)
            ENDWHILE
         ;ENDFOLD (Check that the Nut Feeder is Home)
         bGunReady2Start=bGunReady2Start AND dipw_SpearHome(nutweldINFO.GunNr) AND NOT bSkipFdrHmChk
         SWITCH nutweldINFO.GunNr
            CASE 1
               WAIT FOR bpw1_GunAtHome AND NOT bpw1_GunAtWork
               bGunReady2Start=bGunReady2Start AND bpw1_GunAtHome AND NOT bpw1_GunAtWork
            CASE 2
               WAIT FOR bpw2_GunAtHome AND NOT bpw2_GunAtWork
               bGunReady2Start=bGunReady2Start AND bpw2_GunAtHome AND NOT bpw2_GunAtWork
            CASE 3
               WAIT FOR bpw3_GunAtHome AND NOT bpw3_GunAtWork
               bGunReady2Start=bGunReady2Start AND bpw3_GunAtHome AND NOT bpw3_GunAtWork
         ENDSWITCH
         WAIT FOR dipw_XtfmrTempOk(nutweldINFO.GunNr)
         WAIT FOR dipw_WaterOk(nutweldINFO.GunNr)
         WAIT FOR dipw_WaterTempOk(nutweldINFO.GunNr)
         WAIT FOR NOT dipw_IntensfPresOk(nutweldINFO.GunNr)
         WAIT FOR dipw_Ready(nutweldINFO.GunNr)
         WAIT FOR NOT dipw_Fault(nutweldINFO.GunNr)
         WAIT FOR dipw_SpearHome(nutweldINFO.GunNr)
         WAIT FOR bGunReady2Start AND dipw_XtfmrTempOk(nutweldINFO.GunNr) AND dipw_WaterOk(nutweldINFO.GunNr) AND dipw_WaterTempOk(nutweldINFO.GunNr) AND NOT dipw_IntensfPresOk(nutweldINFO.GunNr) AND dipw_Ready(nutweldINFO.GunNr) AND NOT dipw_Fault(nutweldINFO.GunNr) AND dipw_SpearHome(nutweldINFO.GunNr)
         eCurrentState=#Wait2Weld
      ;ENDFOLD (Implementation)
   ;ENDFOLD (Details)
END ; (PreNutWeldSup)

DEF OpenNutGun(nutweldINFO :IN )
   ;FOLD Details
      ;FOLD Declaration
         DECL NutWeldDAT nutweldINFO
         DECL BOOL bSkipOpenChk
         DECL BOOL bMsgRelease
      ;ENDFOLD (Declaration)
      ;FOLD Implementation
         bMsgRelease=FALSE
         bSkipOpenChk=FALSE
         dopw_BlowOff(nutweldINFO.GunNr,FALSE)
         dopw_NutIntensify(nutweldINFO.GunNr,FALSE)
         ;FOLD TimeOut Setup
            $TIMER_STOP[nNutWeldSignalTmr]=TRUE
            $TIMER[nNutWeldSignalTmr]=nNutWeld_Signal_Timeout*(-1)
            $TIMER_STOP[nNutWeldSignalTmr]=FALSE
         ;ENDFOLD (TimeOut Setup)
         WAIT FOR ((dipw_IntensfPresOk(nutweldINFO.GunNr)==FALSE) OR ($TIMER_FLAG[nNutWeldSignalTmr]==TRUE))
         $TIMER_STOP[nNutWeldSignalTmr]=TRUE
         WHILE ((dipw_IntensfPresOk(nutweldINFO.GunNr)==TRUE) AND (bSkipOpenChk==FALSE))
            ;FOLD Dialog "Nut Welder Intensify Pressure Fault!  Pressure Switch Remained On From Last Cycle!"
               REPEAT
                  nNutWeld_Handle = Set_KrlDlg (NutWeld_Msg[17], NutWeld_MsgPar[], NutWeld_SK_RetrySkip[], NutWeld_MsgOpt_Stop)
                  IF (nNutWeld_Handle > 0) THEN
                     WHILE (Exists_KrlDlg(nNutWeld_Handle, nNutWeld_Key))
                        IF ($ERR.Int_Prio>0) THEN
                           BRAKE
                        ENDIF
                        WAIT SEC 0.024
                     ENDWHILE
                     SWITCH nNutWeld_Key
                        CASE 1 ; Diagnostic
                           nNutWeld_Handle = Set_Krlmsg (#QUIT, NutWeld_Msg[2], NutWeld_MsgPar[], NutWeld_MsgOpt_Stop)
                           WHILE (Exists_KrlMsg(nNutWeld_Handle))
                              WAIT SEC 0.024
                           ENDWHILE
                        CASE 2 ; Retry
                           bMsgRelease=TRUE
                           ;FOLD TimeOut Setup
                              $TIMER_STOP[nNutWeldSignalTmr]=TRUE
                              $TIMER[nNutWeldSignalTmr]=nNutWeld_Signal_Timeout*(-1)
                              $TIMER_STOP[nNutWeldSignalTmr]=FALSE
                           ;ENDFOLD (TimeOut Setup)
                           WAIT FOR ((dipw_IntensfPresOk(nutweldINFO.GunNr)==FALSE) OR ($TIMER_FLAG[nNutWeldSignalTmr]==TRUE))
                        CASE 3 ; Skip
                           WAIT SEC 0.100
                           bMsgRelease=TRUE
                           bSkipOpenChk=TRUE
                     ENDSWITCH
                  ENDIF
               UNTIL (bMsgRelease==TRUE)
               bMsgRelease=FALSE
            ;ENDFOLD (Dialog)
         ENDWHILE
         bSkipOpenChk=FALSE
         dopw_GunWork(nutweldINFO.GunNr,FALSE)
         ;FOLD Wait for Gun At Home
            WHILE ((bNutWeldWOJoining==FALSE) AND (bpw_GunAtHome(nutweldINFO.GunNr )==FALSE) AND (bSkipOpenChk==FALSE))
               $TIMER_STOP[nNutWeldSignalTmr]=TRUE
               $TIMER[nNutWeldSignalTmr]=nNutWeld_Signal_Timeout*(-1)
               $TIMER_STOP[nNutWeldSignalTmr]=FALSE
               WAIT FOR (((bpw_GunAtHome(nutweldINFO.GunNr)==TRUE) AND (bpw_GunAtWork(nutweldINFO.GunNr)==FALSE)) OR ($TIMER_FLAG[nNutWeldSignalTmr]==TRUE))
               $TIMER_STOP[nNutWeldSignalTmr]=TRUE
               IF (bpw_GunAtHome(nutweldINFO.GunNr)==FALSE) THEN
                  ;FOLD Dialog "Nut Welder Open Switch Fault!  Open Switch is not ON!"
                     REPEAT
                        nNutWeld_Handle = Set_KrlDlg (NutWeld_Msg[3], NutWeld_MsgPar[], NutWeld_SK_RetrySkip[], NutWeld_MsgOpt_Stop)
                        IF (nNutWeld_Handle > 0) THEN
                           WHILE (Exists_KrlDlg(nNutWeld_Handle, nNutWeld_Key))
                              WAIT SEC 0.024
                           ENDWHILE
                           SWITCH nNutWeld_Key
                              CASE 1 ; Diagnostic
                                 nNutWeld_Handle = Set_Krlmsg (#QUIT, NutWeld_Msg[2], NutWeld_MsgPar[], NutWeld_MsgOpt_Stop)
                                 WHILE (Exists_KrlMsg(nNutWeld_Handle))
                                    WAIT SEC 0.024
                                 ENDWHILE
                              CASE 2 ; Retry
                                 dopw_GunWork(nutweldINFO.GunNr,FALSE)
                                 bMsgRelease=TRUE
                              CASE 3 ; Skip
                                 WAIT SEC 0.100
                                 bMsgRelease=TRUE
                                 bSkipOpenChk=TRUE
                           ENDSWITCH
                        ENDIF
                     UNTIL (bMsgRelease==TRUE)
                     bMsgRelease=FALSE
                  ;ENDFOLD (Dialog)
               ELSE
                  IF (bpw_GunAtWork(nutweldINFO.GunNr)==TRUE) THEN
                     ;FOLD Dialog "Nut Welder Close Switch Fault!  Close Switch is not OFF!"
                        REPEAT
                           nNutWeld_Handle = Set_KrlDlg (NutWeld_Msg[46], NutWeld_MsgPar[], NutWeld_SK_RetrySkip[], NutWeld_MsgOpt_Stop)
                           IF (nNutWeld_Handle > 0) THEN
                              WHILE (Exists_KrlDlg(nNutWeld_Handle, nNutWeld_Key))
                                 WAIT SEC 0.024
                              ENDWHILE
                              SWITCH nNutWeld_Key
                                 CASE 1 ; Diagnostic
                                    nNutWeld_Handle = Set_Krlmsg (#QUIT, NutWeld_Msg[2], NutWeld_MsgPar[], NutWeld_MsgOpt_Stop)
                                    WHILE (Exists_KrlMsg(nNutWeld_Handle))
                                       WAIT SEC 0.024
                                    ENDWHILE
                                 CASE 2 ; Retry
                                    dopw_GunWork(nutweldINFO.GunNr,FALSE)
                                    bMsgRelease=TRUE
                                 CASE 3 ; Skip
                                    WAIT SEC 0.100
                                    bMsgRelease=TRUE
                                    bSkipOpenChk=TRUE
                              ENDSWITCH
                           ENDIF
                        UNTIL (bMsgRelease==TRUE)
                        bMsgRelease=FALSE
                     ;ENDFOLD (Dialog)
                  ENDIF
               ENDIF
            ENDWHILE
            bSkipOpenChk=FALSE
         ;ENDFOLD (Wait for Gun At Home)
      ;ENDFOLD (Implementation)
   ;ENDFOLD (Details)
END ; (OpenNutGun)

